LIN {X 0,Y 467.594,Z 130.241,A -85,B 0,C 180,E1 -7494.888,E2 -7494.888} C_VEL
LIN {X 0,Y 467.619,Z 130.232,A -85,B 0,C 180,E1 -7497.769,E2 -7497.769} C_VEL
LIN {X 0,Y 467.567,Z 130.241,A -85,B 0,C 180,E1 -7501.045,E2 -7501.045} C_VEL
LIN {X 0,Y 467.576,Z 130.242,A -85,B 0,C 180,E1 -7504.24,E2 -7504.24} C_VEL
LIN {X 0,Y 467.547,Z 130.241,A -85,B 0,C 180,E1 -7507.186,E2 -7507.186} C_VEL
LIN {X 0,Y 467.573,Z 130.245,A -85,B 0,C 180,E1 -7510.265,E2 -7510.265} C_VEL
LIN {X 0,Y 467.585,Z 130.24,A -85,B 0,C 180,E1 -7512.567,E2 -7512.567} C_VEL
LIN {X 0,Y 467.569,Z 130.238,A -85,B 0,C 180,E1 -7515.053,E2 -7515.053} C_VEL
LIN {X 0,Y 467.587,Z 130.236,A -85,B 0,C 180,E1 -7517.44,E2 -7517.44} C_VEL
LIN {X 0,Y 467.581,Z 130.237,A -85,B 0,C 180,E1 -7520.855,E2 -7520.855} C_VEL
LIN {X 0,Y 467.56,Z 130.244,A -85,B 0,C 180,E1 -7524.26,E2 -7524.26} C_VEL
LIN {X 0,Y 467.58,Z 130.238,A -85,B 0,C 180,E1 -7527.321,E2 -7527.321} C_VEL
LIN {X 0,Y 467.569,Z 130.238,A -85,B 0,C 180,E1 -7530.667,E2 -7530.667} C_VEL
LIN {X 0,Y 467.611,Z 130.234,A -85,B 0,C 180,E1 -7533.2,E2 -7533.2} C_VEL
LIN {X 0,Y 467.588,Z 130.236,A -85,B 0,C 180,E1 -7536.469,E2 -7536.469} C_VEL
LIN {X 0,Y 467.621,Z 130.237,A -85,B 0,C 180,E1 -7539.777,E2 -7539.777} C_VEL
LIN {X 0,Y 467.607,Z 130.233,A -85,B 0,C 180,E1 -7542.507,E2 -7542.507} C_VEL
LIN {X 0,Y 467.608,Z 130.238,A -85,B 0,C 180,E1 -7545.197,E2 -7545.197} C_VEL
LIN {X 0,Y 467.654,Z 130.23,A -85,B 0,C 180,E1 -7547.855,E2 -7547.855} C_VEL
LIN {X 0,Y 467.68,Z 130.232,A -85,B 0,C 180,E1 -7551.357,E2 -7551.357} C_VEL
LIN {X 0,Y 467.744,Z 130.217,A -85,B 0,C 180,E1 -7553.963,E2 -7553.963} C_VEL
LIN {X 0,Y 467.858,Z 130.207,A -85,B 0,C 180,E1 -7557.417,E2 -7557.417} C_VEL
LIN {X 0,Y 467.881,Z 130.199,A -85,B 0,C 180,E1 -7560,E2 -7560} C_VEL
LIN {X 0,Y 467.858,Z 130.204,A -85,B 0,C 180,E1 -7562.583,E2 -7562.583} C_VEL
LIN {X 0,Y 467.734,Z 130.218,A -85,B 0,C 180,E1 -7566.038,E2 -7566.038} C_VEL
LIN {X 0,Y 467.68,Z 130.229,A -85,B 0,C 180,E1 -7568.643,E2 -7568.643} C_VEL
LIN {X 0,Y 467.655,Z 130.228,A -85,B 0,C 180,E1 -7572.146,E2 -7572.146} C_VEL
LIN {X 0,Y 467.638,Z 130.229,A -85,B 0,C 180,E1 -7575.695,E2 -7575.695} C_VEL
LIN {X 0,Y 467.617,Z 130.238,A -85,B 0,C 180,E1 -7578.765,E2 -7578.765} C_VEL
LIN {X 0,Y 467.579,Z 130.238,A -85,B 0,C 180,E1 -7581.268,E2 -7581.268} C_VEL
LIN {X 0,Y 467.571,Z 130.239,A -85,B 0,C 180,E1 -7583.944,E2 -7583.944} C_VEL
LIN {X 0,Y 467.616,Z 130.236,A -85,B 0,C 180,E1 -7586.801,E2 -7586.801} C_VEL
LIN {X 0,Y 467.553,Z 130.241,A -85,B 0,C 180,E1 -7589.738,E2 -7589.738} C_VEL
LIN {X 0,Y 467.583,Z 130.239,A -85,B 0,C 180,E1 -7592.759,E2 -7592.759} C_VEL
LIN {X 0,Y 467.553,Z 130.244,A -85,B 0,C 180,E1 -7595.89,E2 -7595.89} C_VEL
LIN {X 0,Y 467.6,Z 130.234,A -85,B 0,C 180,E1 -7599.143,E2 -7599.143} C_VEL
LIN {X 0,Y 467.587,Z 130.238,A -85,B 0,C 180,E1 -7602.567,E2 -7602.567} C_VEL
LIN {X 0,Y 467.571,Z 130.238,A -85,B 0,C 180,E1 -7605.053,E2 -7605.053} C_VEL
LIN {X 0,Y 467.59,Z 130.238,A -85,B 0,C 180,E1 -7607.44,E2 -7607.44} C_VEL
LIN {X 0,Y 467.601,Z 130.234,A -85,B 0,C 180,E1 -7610.857,E2 -7610.857} C_VEL
LIN {X 0,Y 467.561,Z 130.241,A -85,B 0,C 180,E1 -7614.261,E2 -7614.261} C_VEL
LIN {X 0,Y 467.583,Z 130.24,A -85,B 0,C 180,E1 -7617.321,E2 -7617.321} C_VEL
LIN {X 0,Y 467.572,Z 130.242,A -85,B 0,C 180,E1 -7620.668,E2 -7620.668} C_VEL
LIN {X 0,Y 467.701,Z 130.331,A -85,B 0,C 180,E1 -7623.093,E2 -7623.093} C_VEL
LIN {X 0,Y 470,Z 142.281,A -85,B 0,C 180,E1 -7625.248,E2 -7625.248} C_VEL
LIN {X 0,Y 469.567,Z 154.773,A -85,B 0,C 180,E1 -7627.332,E2 -7627.332} C_VEL
LIN {X 0,Y 468.805,Z 175.972,A -85,B 0,C 180,E1 -7630.814,E2 -7630.814} C_VEL
LIN {X 0,Y 468.241,Z 189.54,A -85,B 0,C 180,E1 -7633.002,E2 -7633.002} C_VEL
LIN {X 0,Y 471.063,Z 210.719,A -85,B 0,C 180,E1 -7633.441,E2 -7633.441} C_VEL
LIN {X 0,Y 470.388,Z 298.839,A -85,B 0,C 180,E1 -7634.843,E2 -7634.843} C_VEL
LIN {X 0,Y 469.978,Z 311.849,A -85,B 0,C 180,E1 -7635.218,E2 -7635.218} C_VEL
LIN {X 0,Y 469.486,Z 324.472,A -85,B 0,C 180,E1 -7635.755,E2 -7635.755} C_VEL
LIN {X 0,Y 469.009,Z 336.521,A -85,B 0,C 180,E1 -7636.459,E2 -7636.459} C_VEL
LIN {X 0,Y 468.479,Z 348.326,A -85,B 0,C 180,E1 -7637.35,E2 -7637.35} C_VEL
LIN {X 0,Y 468.04,Z 358.45,A -85,B 0,C 180,E1 -7638.304,E2 -7638.304} C_VEL
LIN {X 0,Y 467.56,Z 367.788,A -85,B 0,C 180,E1 -7639.389,E2 -7639.389} C_VEL
LIN {X 0,Y 467.188,Z 376.856,A -85,B 0,C 180,E1 -7640.694,E2 -7640.694} C_VEL
LIN {X 0,Y 466.977,Z 384.164,A -85,B 0,C 180,E1 -7641.998,E2 -7641.998} C_VEL
LIN {X 0,Y 466.827,Z 389.097,A -85,B 0,C 180,E1 -7643.083,E2 -7643.083} C_VEL
LIN {X 0,Y 466.746,Z 393.889,A -85,B 0,C 180,E1 -7644.383,E2 -7644.383} C_VEL
LIN {X 0,Y 466.659,Z 397.547,A -85,B 0,C 180,E1 -7645.681,E2 -7645.681} C_VEL
LIN {X 0,Y 466.747,Z 399.441,A -85,B 0,C 180,E1 -7646.547,E2 -7646.547} C_VEL
LIN {X 0,Y 466.711,Z 400.855,A -85,B 0,C 180,E1 -7647.411,E2 -7647.411} C_VEL
LIN {X 0,Y 466.696,Z 401.858,A -85,B 0,C 180,E1 -7648.274,E2 -7648.274} C_VEL
LIN {X 0,Y 466.621,Z 402.678,A -85,B 0,C 180,E1 -7650,E2 -7650} C_VEL
LIN {X 0,Y 466.634,Z 402.453,A -85,B 0,C 180,E1 -7650.863,E2 -7650.863} C_VEL
LIN {X 0,Y 466.696,Z 401.831,A -85,B 0,C 180,E1 -7651.726,E2 -7651.726} C_VEL
LIN {X 0,Y 466.711,Z 400.812,A -85,B 0,C 180,E1 -7652.589,E2 -7652.589} C_VEL
LIN {X 0,Y 466.748,Z 399.388,A -85,B 0,C 180,E1 -7653.453,E2 -7653.453} C_VEL
LIN {X 0,Y 466.689,Z 396.392,A -85,B 0,C 180,E1 -7654.751,E2 -7654.751} C_VEL
LIN {X 0,Y 466.713,Z 392.348,A -85,B 0,C 180,E1 -7656.051,E2 -7656.051} C_VEL
LIN {X 0,Y 466.904,Z 386.14,A -85,B 0,C 180,E1 -7657.568,E2 -7657.568} C_VEL
LIN {X 0,Y 467.077,Z 379.359,A -85,B 0,C 180,E1 -7658.872,E2 -7658.872} C_VEL
LIN {X 0,Y 467.396,Z 370.96,A -85,B 0,C 180,E1 -7660.176,E2 -7660.176} C_VEL
LIN {X 0,Y 467.834,Z 362.352,A -85,B 0,C 180,E1 -7661.262,E2 -7661.262} C_VEL
LIN {X 0,Y 468.252,Z 352.515,A -85,B 0,C 180,E1 -7662.277,E2 -7662.277} C_VEL
LIN {X 0,Y 468.773,Z 341.227,A -85,B 0,C 180,E1 -7663.216,E2 -7663.216} C_VEL
LIN {X 0,Y 469.307,Z 329.707,A -85,B 0,C 180,E1 -7663.974,E2 -7663.974} C_VEL
LIN {X 0,Y 469.764,Z 317.81,A -85,B 0,C 180,E1 -7664.568,E2 -7664.568} C_VEL
LIN {X 0,Y 470.275,Z 304.132,A -85,B 0,C 180,E1 -7665.05,E2 -7665.05} C_VEL
LIN {X 0,Y 470.563,Z 290.188,A -85,B 0,C 180,E1 -7665.345,E2 -7665.345} C_VEL
LIN {X 0,Y 471.015,Z 208.612,A -85,B 0,C 180,E1 -7666.634,E2 -7666.634} C_VEL
LIN {X 0,Y 468.224,Z 188.606,A -85,B 0,C 180,E1 -7667.064,E2 -7667.064} C_VEL
LIN {X 0,Y 468.823,Z 169.364,A -85,B 0,C 180,E1 -7670.169,E2 -7670.169} C_VEL
LIN {X 0,Y 469.527,Z 152.566,A -85,B 0,C 180,E1 -7672.903,E2 -7672.903} C_VEL
LIN {X 0,Y 469.89,Z 142.442,A -85,B 0,C 180,E1 -7674.575,E2 -7674.575} C_VEL
LIN {X 0,Y 468.192,Z 132.826,A -85,B 0,C 180,E1 -7676.283,E2 -7676.283} C_VEL
LIN {X 0,Y 467.673,Z 130.234,A -85,B 0,C 180,E1 -7676.797,E2 -7676.797} C_VEL
LIN {X 0,Y 467.556,Z 130.246,A -85,B 0,C 180,E1 -7679.738,E2 -7679.738} C_VEL
LIN {X 0,Y 467.584,Z 130.242,A -85,B 0,C 180,E1 -7682.758,E2 -7682.758} C_VEL
LIN {X 0,Y 467.554,Z 130.246,A -85,B 0,C 180,E1 -7685.889,E2 -7685.889} C_VEL
LIN {X 0,Y 467.601,Z 130.238,A -85,B 0,C 180,E1 -7689.143,E2 -7689.143} C_VEL
LIN {X 0,Y 467.587,Z 130.241,A -85,B 0,C 180,E1 -7692.567,E2 -7692.567} C_VEL
LIN {X 0,Y 467.57,Z 130.241,A -85,B 0,C 180,E1 -7695.053,E2 -7695.053} C_VEL
LIN {X 0,Y 467.589,Z 130.24,A -85,B 0,C 180,E1 -7697.44,E2 -7697.44} C_VEL
LIN {X 0,Y 467.599,Z 130.234,A -85,B 0,C 180,E1 -7700.857,E2 -7700.857} C_VEL
LIN {X 0,Y 467.559,Z 130.243,A -85,B 0,C 180,E1 -7704.261,E2 -7704.261} C_VEL
LIN {X 0,Y 467.581,Z 130.238,A -85,B 0,C 180,E1 -7707.321,E2 -7707.321} C_VEL
LIN {X 0,Y 467.568,Z 130.236,A -85,B 0,C 180,E1 -7710.667,E2 -7710.667} C_VEL
LIN {X 0,Y 467.612,Z 130.235,A -85,B 0,C 180,E1 -7713.199,E2 -7713.199} C_VEL
LIN {X 0,Y 467.589,Z 130.234,A -85,B 0,C 180,E1 -7716.468,E2 -7716.468} C_VEL
LIN {X 0,Y 467.622,Z 130.234,A -85,B 0,C 180,E1 -7719.777,E2 -7719.777} C_VEL
LIN {X 0,Y 467.607,Z 130.233,A -85,B 0,C 180,E1 -7722.506,E2 -7722.506} C_VEL
LIN {X 0,Y 467.608,Z 130.235,A -85,B 0,C 180,E1 -7725.196,E2 -7725.196} C_VEL
LIN {X 0,Y 467.654,Z 130.228,A -85,B 0,C 180,E1 -7727.854,E2 -7727.854} C_VEL
LIN {X 0,Y 467.68,Z 130.229,A -85,B 0,C 180,E1 -7731.357,E2 -7731.357} C_VEL
LIN {X 0,Y 467.744,Z 130.218,A -85,B 0,C 180,E1 -7733.962,E2 -7733.962} C_VEL
LIN {X 0,Y 467.858,Z 130.207,A -85,B 0,C 180,E1 -7737.417,E2 -7737.417} C_VEL
LIN {X 0,Y 467.881,Z 130.198,A -85,B 0,C 180,E1 -7740,E2 -7740} C_VEL
LIN {X 0,Y 467.858,Z 130.206,A -85,B 0,C 180,E1 -7742.583,E2 -7742.583} C_VEL
LIN {X 0,Y 467.733,Z 130.217,A -85,B 0,C 180,E1 -7746.037,E2 -7746.037} C_VEL
LIN {X 0,Y 467.679,Z 130.231,A -85,B 0,C 180,E1 -7748.643,E2 -7748.643} C_VEL
LIN {X 0,Y 467.654,Z 130.229,A -85,B 0,C 180,E1 -7752.145,E2 -7752.145} C_VEL
LIN {X 0,Y 467.637,Z 130.231,A -85,B 0,C 180,E1 -7755.695,E2 -7755.695} C_VEL
LIN {X 0,Y 467.615,Z 130.24,A -85,B 0,C 180,E1 -7758.765,E2 -7758.765} C_VEL
LIN {X 0,Y 467.578,Z 130.239,A -85,B 0,C 180,E1 -7761.268,E2 -7761.268} C_VEL
LIN {X 0,Y 467.569,Z 130.244,A -85,B 0,C 180,E1 -7763.943,E2 -7763.943} C_VEL
LIN {X 0,Y 467.614,Z 130.24,A -85,B 0,C 180,E1 -7766.8,E2 -7766.8} C_VEL
LIN {X 0,Y 467.552,Z 130.244,A -85,B 0,C 180,E1 -7769.738,E2 -7769.738} C_VEL
LIN {X 0,Y 467.582,Z 130.244,A -85,B 0,C 180,E1 -7772.758,E2 -7772.758} C_VEL
LIN {X 0,Y 467.651,Z 130.325,A -85,B 0,C 180,E1 -7773.589,E2 -7773.589} C_VEL
LIN {X 0,Y 468.729,Z 136.861,A -85,B 0,C 180,E1 -7774.995,E2 -7774.995} C_VEL
LIN {X 0,Y 468.69,Z 141.798,A -85,B 0,C 180,E1 -7776.011,E2 -7776.011} C_VEL
LIN {X 0,Y 471.496,Z 154.916,A -85,B 0,C 180,E1 -7776.345,E2 -7776.345} C_VEL
LIN {X 0,Y 470.667,Z 248.936,A -85,B 0,C 180,E1 -7777.851,E2 -7777.851} C_VEL
LIN {X 0,Y 470.374,Z 262.577,A -85,B 0,C 180,E1 -7778.252,E2 -7778.252} C_VEL
LIN {X 0,Y 470.103,Z 274.187,A -85,B 0,C 180,E1 -7778.757,E2 -7778.757} C_VEL
LIN {X 0,Y 469.739,Z 285.551,A -85,B 0,C 180,E1 -7779.414,E2 -7779.414} C_VEL
LIN {X 0,Y 469.285,Z 296.959,A -85,B 0,C 180,E1 -7780.267,E2 -7780.267} C_VEL
LIN {X 0,Y 468.755,Z 307.729,A -85,B 0,C 180,E1 -7781.276,E2 -7781.276} C_VEL
LIN {X 0,Y 468.315,Z 316.44,A -85,B 0,C 180,E1 -7782.282,E2 -7782.282} C_VEL
LIN {X 0,Y 467.855,Z 325.055,A -85,B 0,C 180,E1 -7783.503,E2 -7783.503} C_VEL
LIN {X 0,Y 467.497,Z 332.108,A -85,B 0,C 180,E1 -7784.737,E2 -7784.737} C_VEL
LIN {X 0,Y 467.196,Z 338.877,A -85,B 0,C 180,E1 -7786.225,E2 -7786.225} C_VEL
LIN {X 0,Y 467.002,Z 343.41,A -85,B 0,C 180,E1 -7787.511,E2 -7787.511} C_VEL
LIN {X 0,Y 466.836,Z 346.943,A -85,B 0,C 180,E1 -7788.827,E2 -7788.827} C_VEL
LIN {X 0,Y 466.724,Z 349.492,A -85,B 0,C 180,E1 -7790.171,E2 -7790.171} C_VEL
LIN {X 0,Y 466.622,Z 351.29,A -85,B 0,C 180,E1 -7791.919,E2 -7791.919} C_VEL
LIN {X 0,Y 466.617,Z 351.63,A -85,B 0,C 180,E1 -7792.964,E2 -7792.964} C_VEL
LIN {X 0,Y 466.608,Z 351.1,A -85,B 0,C 180,E1 -7794.424,E2 -7794.424} C_VEL
LIN {X 0,Y 466.69,Z 349.689,A -85,B 0,C 180,E1 -7795.672,E2 -7795.672} C_VEL
LIN {X 0,Y 466.103,Z 348.636,A -85,B 0,C 180,E1 -7796.383,E2 -7796.383} C_VEL
LIN {X 0,Y 463.361,Z 346.465,A -85,B 0,C 180,E1 -7797.529,E2 -7797.529} C_VEL
LIN {X 0,Y 461.039,Z 344.188,A -85,B 0,C 180,E1 -7798.432,E2 -7798.432} C_VEL
LIN {X 0,Y 460.075,Z 342.059,A -85,B 0,C 180,E1 -7799.112,E2 -7799.112} C_VEL
LIN {X 0,Y 460.016,Z 341.258,A -85,B 0,C 180,E1 -7799.338,E2 -7799.338} C_VEL
LIN {X 0,Y 460.283,Z 335.541,A -85,B 0,C 180,E1 -7800.751,E2 -7800.751} C_VEL
LIN {X 0,Y 460.683,Z 327.924,A -85,B 0,C 180,E1 -7802.23,E2 -7802.23} C_VEL
LIN {X 0,Y 461.124,Z 319.458,A -85,B 0,C 180,E1 -7803.526,E2 -7803.526} C_VEL
LIN {X 0,Y 461.649,Z 309.352,A -85,B 0,C 180,E1 -7804.77,E2 -7804.77} C_VEL
LIN {X 0,Y 462.112,Z 299.402,A -85,B 0,C 180,E1 -7805.756,E2 -7805.756} C_VEL
LIN {X 0,Y 462.609,Z 288.553,A -85,B 0,C 180,E1 -7806.616,E2 -7806.616} C_VEL
LIN {X 0,Y 463.013,Z 276.885,A -85,B 0,C 180,E1 -7807.346,E2 -7807.346} C_VEL
LIN {X 0,Y 463.364,Z 265.358,A -85,B 0,C 180,E1 -7807.894,E2 -7807.894} C_VEL
LIN {X 0,Y 463.657,Z 252.665,A -85,B 0,C 180,E1 -7808.317,E2 -7808.317} C_VEL
LIN {X 0,Y 463.828,Z 237.232,A -85,B 0,C 180,E1 -7808.617,E2 -7808.617} C_VEL
LIN {X 0,Y 464.471,Z 155.674,A -85,B 0,C 180,E1 -7809.919,E2 -7809.919} C_VEL
LIN {X 0,Y 461.531,Z 141.472,A -85,B 0,C 180,E1 -7810.279,E2 -7810.279} C_VEL
LIN {X 0,Y 461.356,Z 135.46,A -85,B 0,C 180,E1 -7811.573,E2 -7811.573} C_VEL
LIN {X 0,Y 460.578,Z 131.114,A -85,B 0,C 180,E1 -7812.575,E2 -7812.575} C_VEL
LIN {X 0,Y 460.565,Z 131.114,A -85,B 0,C 180,E1 -7814.965,E2 -7814.965} C_VEL
LIN {X 0,Y 460.61,Z 131.105,A -85,B 0,C 180,E1 -7818.559,E2 -7818.559} C_VEL
LIN {X 0,Y 460.695,Z 131.096,A -85,B 0,C 180,E1 -7822.109,E2 -7822.109} C_VEL
LIN {X 0,Y 460.695,Z 131.095,A -85,B 0,C 180,E1 -7824.748,E2 -7824.748} C_VEL
LIN {X 0,Y 460.799,Z 131.089,A -85,B 0,C 180,E1 -7827.378,E2 -7827.378} C_VEL
LIN {X 0,Y 460.853,Z 131.076,A -85,B 0,C 180,E1 -7830,E2 -7830} C_VEL
LIN {X 0,Y 460.8,Z 131.082,A -85,B 0,C 180,E1 -7832.623,E2 -7832.623} C_VEL
LIN {X 0,Y 460.688,Z 131.095,A -85,B 0,C 180,E1 -7836.13,E2 -7836.13} C_VEL
LIN {X 0,Y 460.619,Z 131.107,A -85,B 0,C 180,E1 -7838.776,E2 -7838.776} C_VEL
LIN {X 0,Y 460.614,Z 131.106,A -85,B 0,C 180,E1 -7842.445,E2 -7842.445} C_VEL
LIN {X 0,Y 460.6,Z 131.106,A -85,B 0,C 180,E1 -7845.997,E2 -7845.997} C_VEL
LIN {X 0,Y 460.568,Z 131.111,A -85,B 0,C 180,E1 -7849.615,E2 -7849.615} C_VEL
LIN {X 0,Y 460.51,Z 131.121,A -85,B 0,C 180,E1 -7852.429,E2 -7852.429} C_VEL
LIN {X 0,Y 460.557,Z 131.112,A -85,B 0,C 180,E1 -7855.799,E2 -7855.799} C_VEL
LIN {X 0,Y 460.552,Z 131.115,A -85,B 0,C 180,E1 -7858.233,E2 -7858.233} C_VEL
LIN {X 0,Y 460.519,Z 131.117,A -85,B 0,C 180,E1 -7861.283,E2 -7861.283} C_VEL
LIN {X 0,Y 460.522,Z 131.124,A -85,B 0,C 180,E1 -7864.504,E2 -7864.504} C_VEL
LIN {X 0,Y 460.5,Z 131.119,A -85,B 0,C 180,E1 -7867.623,E2 -7867.623} C_VEL
LIN {X 0,Y 460.537,Z 131.121,A -85,B 0,C 180,E1 -7870.269,E2 -7870.269} C_VEL
LIN {X 0,Y 460.498,Z 131.119,A -85,B 0,C 180,E1 -7873.375,E2 -7873.375} C_VEL
LIN {X 0,Y 460.498,Z 131.122,A -85,B 0,C 180,E1 -7876.625,E2 -7876.625} C_VEL
LIN {X 0,Y 460.54,Z 131.117,A -85,B 0,C 180,E1 -7879.731,E2 -7879.731} C_VEL
LIN {X 0,Y 460.525,Z 131.118,A -85,B 0,C 180,E1 -7882.519,E2 -7882.519} C_VEL
LIN {X 0,Y 460.546,Z 131.117,A -85,B 0,C 180,E1 -7885.624,E2 -7885.624} C_VEL
LIN {X 0,Y 460.535,Z 131.114,A -85,B 0,C 180,E1 -7888.745,E2 -7888.745} C_VEL
LIN {X 0,Y 460.579,Z 131.111,A -85,B 0,C 180,E1 -7892.254,E2 -7892.254} C_VEL
LIN {X 0,Y 460.537,Z 131.114,A -85,B 0,C 180,E1 -7894.704,E2 -7894.704} C_VEL
LIN {X 0,Y 460.508,Z 131.124,A -85,B 0,C 180,E1 -7897.571,E2 -7897.571} C_VEL
LIN {X 0,Y 460.567,Z 131.111,A -85,B 0,C 180,E1 -7900.385,E2 -7900.385} C_VEL
LIN {X 0,Y 460.563,Z 131.114,A -85,B 0,C 180,E1 -7903.146,E2 -7903.146} C_VEL
LIN {X 0,Y 460.556,Z 131.115,A -85,B 0,C 180,E1 -7905.868,E2 -7905.868} C_VEL
LIN {X 0,Y 460.61,Z 131.105,A -85,B 0,C 180,E1 -7908.559,E2 -7908.559} C_VEL
LIN {X 0,Y 460.694,Z 131.095,A -85,B 0,C 180,E1 -7912.109,E2 -7912.109} C_VEL
LIN {X 0,Y 460.697,Z 131.096,A -85,B 0,C 180,E1 -7914.749,E2 -7914.749} C_VEL
LIN {X 0,Y 460.823,Z 131.084,A -85,B 0,C 180,E1 -7917.378,E2 -7917.378} C_VEL
LIN {X 0,Y 460.852,Z 131.075,A -85,B 0,C 180,E1 -7920,E2 -7920} C_VEL
LIN {X 0,Y 460.823,Z 131.081,A -85,B 0,C 180,E1 -7922.623,E2 -7922.623} C_VEL
LIN {X 0,Y 460.7,Z 131.094,A -85,B 0,C 180,E1 -7926.13,E2 -7926.13} C_VEL
LIN {X 0,Y 460.627,Z 131.109,A -85,B 0,C 180,E1 -7928.776,E2 -7928.776} C_VEL
LIN {X 0,Y 460.612,Z 131.108,A -85,B 0,C 180,E1 -7932.445,E2 -7932.445} C_VEL
LIN {X 0,Y 460.599,Z 131.107,A -85,B 0,C 180,E1 -7935.998,E2 -7935.998} C_VEL
LIN {X 0,Y 460.57,Z 131.114,A -85,B 0,C 180,E1 -7938.902,E2 -7938.902} C_VEL
LIN {X 0,Y 460.515,Z 131.117,A -85,B 0,C 180,E1 -7941.486,E2 -7941.486} C_VEL
LIN {X 0,Y 460.541,Z 131.119,A -85,B 0,C 180,E1 -7944.333,E2 -7944.333} C_VEL
LIN {X 0,Y 460.572,Z 131.11,A -85,B 0,C 180,E1 -7947.244,E2 -7947.244} C_VEL
LIN {X 0,Y 460.51,Z 131.124,A -85,B 0,C 180,E1 -7950.24,E2 -7950.24} C_VEL
LIN {X 0,Y 460.529,Z 131.115,A -85,B 0,C 180,E1 -7953.325,E2 -7953.325} C_VEL
LIN {X 0,Y 460.476,Z 131.125,A -85,B 0,C 180,E1 -7956.53,E2 -7956.53} C_VEL
LIN {X 0,Y 460.575,Z 131.114,A -85,B 0,C 180,E1 -7959.858,E2 -7959.858} C_VEL
LIN {X 0,Y 460.513,Z 131.117,A -85,B 0,C 180,E1 -7962.901,E2 -7962.901} C_VEL
LIN {X 0,Y 460.512,Z 131.123,A -85,B 0,C 180,E1 -7965.831,E2 -7965.831} C_VEL
LIN {X 0,Y 460.54,Z 131.114,A -85,B 0,C 180,E1 -7968.99,E2 -7968.99} C_VEL
LIN {X 0,Y 460.541,Z 131.115,A -85,B 0,C 180,E1 -7971.269,E2 -7971.269} C_VEL
LIN {X 0,Y 460.511,Z 131.117,A -85,B 0,C 180,E1 -7974.555,E2 -7974.555} C_VEL
LIN {X 0,Y 460.533,Z 131.122,A -85,B 0,C 180,E1 -7977.716,E2 -7977.716} C_VEL
LIN {X 0,Y 460.542,Z 131.118,A -85,B 0,C 180,E1 -7980.769,E2 -7980.769} C_VEL
LIN {X 0,Y 460.66,Z 131.23,A -85,B 0,C 180,E1 -7982.885,E2 -7982.885} C_VEL
LIN {X 0,Y 463.022,Z 143.219,A -85,B 0,C 180,E1 -7985.086,E2 -7985.086} C_VEL
LIN {X 0,Y 462.816,Z 151.577,A -85,B 0,C 180,E1 -7986.509,E2 -7986.509} C_VEL
LIN {X 0,Y 462.035,Z 168.201,A -85,B 0,C 180,E1 -7989.289,E2 -7989.289} C_VEL
LIN {X 0,Y 461.526,Z 182.026,A -85,B 0,C 180,E1 -7991.58,E2 -7991.58} C_VEL
LIN {X 0,Y 461.248,Z 189.092,A -85,B 0,C 180,E1 -7992.743,E2 -7992.743} C_VEL
LIN {X 0,Y 464.245,Z 211.74,A -85,B 0,C 180,E1 -7993.221,E2 -7993.221} C_VEL
LIN {X 0,Y 463.532,Z 297.985,A -85,B 0,C 180,E1 -7994.613,E2 -7994.613} C_VEL
LIN {X 0,Y 463.111,Z 311.151,A -85,B 0,C 180,E1 -7994.993,E2 -7994.993} C_VEL
LIN {X 0,Y 462.596,Z 323.858,A -85,B 0,C 180,E1 -7995.539,E2 -7995.539} C_VEL
LIN {X 0,Y 462.055,Z 335.978,A -85,B 0,C 180,E1 -7996.252,E2 -7996.252} C_VEL
LIN {X 0,Y 461.486,Z 347.816,A -85,B 0,C 180,E1 -7997.155,E2 -7997.155} C_VEL
LIN {X 0,Y 461.023,Z 357.967,A -85,B 0,C 180,E1 -7998.124,E2 -7998.124} C_VEL
LIN {X 0,Y 460.557,Z 367.336,A -85,B 0,C 180,E1 -7999.226,E2 -7999.226} C_VEL
LIN {X 0,Y 460.142,Z 376.418,A -85,B 0,C 180,E1 -8000.55,E2 -8000.55} C_VEL
LIN {X 0,Y 459.903,Z 383.737,A -85,B 0,C 180,E1 -8001.874,E2 -8001.874} C_VEL
LIN {X 0,Y 459.74,Z 388.679,A -85,B 0,C 180,E1 -8002.975,E2 -8002.975} C_VEL
LIN {X 0,Y 459.642,Z 393.478,A -85,B 0,C 180,E1 -8004.296,E2 -8004.296} C_VEL
LIN {X 0,Y 459.575,Z 397.145,A -85,B 0,C 180,E1 -8005.615,E2 -8005.615} C_VEL
LIN {X 0,Y 459.642,Z 399.041,A -85,B 0,C 180,E1 -8006.494,E2 -8006.494} C_VEL
LIN {X 0,Y 459.631,Z 400.461,A -85,B 0,C 180,E1 -8007.371,E2 -8007.371} C_VEL
LIN {X 0,Y 459.617,Z 401.467,A -85,B 0,C 180,E1 -8008.247,E2 -8008.247} C_VEL
LIN {X 0,Y 459.551,Z 402.29,A -85,B 0,C 180,E1 -8010,E2 -8010} C_VEL
LIN {X 0,Y 459.566,Z 402.068,A -85,B 0,C 180,E1 -8010.876,E2 -8010.876} C_VEL
LIN {X 0,Y 459.604,Z 401.444,A -85,B 0,C 180,E1 -8011.752,E2 -8011.752} C_VEL
LIN {X 0,Y 459.631,Z 400.426,A -85,B 0,C 180,E1 -8012.629,E2 -8012.629} C_VEL
LIN {X 0,Y 459.642,Z 399.001,A -85,B 0,C 180,E1 -8013.506,E2 -8013.506} C_VEL
LIN {X 0,Y 459.619,Z 396.006,A -85,B 0,C 180,E1 -8014.824,E2 -8014.824} C_VEL
LIN {X 0,Y 459.635,Z 391.248,A -85,B 0,C 180,E1 -8016.342,E2 -8016.342} C_VEL
LIN {X 0,Y 459.865,Z 384.729,A -85,B 0,C 180,E1 -8017.906,E2 -8017.906} C_VEL
LIN {X 0,Y 460.086,Z 377.725,A -85,B 0,C 180,E1 -8019.23,E2 -8019.23} C_VEL
LIN {X 0,Y 460.442,Z 368.969,A -85,B 0,C 180,E1 -8020.554,E2 -8020.554} C_VEL
LIN {X 0,Y 460.95,Z 360.009,A -85,B 0,C 180,E1 -8021.655,E2 -8021.655} C_VEL
LIN {X 0,Y 461.436,Z 349.203,A -85,B 0,C 180,E1 -8022.738,E2 -8022.738} C_VEL
LIN {X 0,Y 461.969,Z 337.843,A -85,B 0,C 180,E1 -8023.639,E2 -8023.639} C_VEL
LIN {X 0,Y 462.586,Z 325.398,A -85,B 0,C 180,E1 -8024.405,E2 -8024.405} C_VEL
LIN {X 0,Y 463.06,Z 313.6,A -85,B 0,C 180,E1 -8024.952,E2 -8024.952} C_VEL
LIN {X 0,Y 463.512,Z 300.871,A -85,B 0,C 180,E1 -8025.359,E2 -8025.359} C_VEL
LIN {X 0,Y 463.773,Z 283.141,A -85,B 0,C 180,E1 -8025.688,E2 -8025.688} C_VEL
LIN {X 0,Y 464.2,Z 209.161,A -85,B 0,C 180,E1 -8026.879,E2 -8026.879} C_VEL
LIN {X 0,Y 461.246,Z 188.093,A -85,B 0,C 180,E1 -8027.356,E2 -8027.356} C_VEL
LIN {X 0,Y 461.892,Z 169.002,A -85,B 0,C 180,E1 -8030.485,E2 -8030.485} C_VEL
LIN {X 0,Y 462.645,Z 152.228,A -85,B 0,C 180,E1 -8033.263,E2 -8033.263} C_VEL
LIN {X 0,Y 462.968,Z 143.686,A -85,B 0,C 180,E1 -8034.698,E2 -8034.698} C_VEL
LIN {X 0,Y 461.199,Z 133.885,A -85,B 0,C 180,E1 -8036.47,E2 -8036.47} C_VEL
LIN {X 0,Y 460.638,Z 131.109,A -85,B 0,C 180,E1 -8036.994,E2 -8036.994} C_VEL
LIN {X 0,Y 460.512,Z 131.125,A -85,B 0,C 180,E1 -8040.24,E2 -8040.24} C_VEL
LIN {X 0,Y 460.53,Z 131.118,A -85,B 0,C 180,E1 -8043.324,E2 -8043.324} C_VEL
LIN {X 0,Y 460.477,Z 131.129,A -85,B 0,C 180,E1 -8046.529,E2 -8046.529} C_VEL
LIN {X 0,Y 460.575,Z 131.117,A -85,B 0,C 180,E1 -8049.857,E2 -8049.857} C_VEL
LIN {X 0,Y 460.513,Z 131.12,A -85,B 0,C 180,E1 -8052.9,E2 -8052.9} C_VEL
LIN {X 0,Y 460.512,Z 131.124,A -85,B 0,C 180,E1 -8055.83,E2 -8055.83} C_VEL
LIN {X 0,Y 460.539,Z 131.115,A -85,B 0,C 180,E1 -8058.989,E2 -8058.989} C_VEL
LIN {X 0,Y 460.539,Z 131.114,A -85,B 0,C 180,E1 -8061.268,E2 -8061.268} C_VEL
LIN {X 0,Y 460.509,Z 131.119,A -85,B 0,C 180,E1 -8064.554,E2 -8064.554} C_VEL
LIN {X 0,Y 460.53,Z 131.119,A -85,B 0,C 180,E1 -8067.715,E2 -8067.715} C_VEL
LIN {X 0,Y 460.538,Z 131.112,A -85,B 0,C 180,E1 -8070.769,E2 -8070.769} C_VEL
LIN {X 0,Y 460.555,Z 131.115,A -85,B 0,C 180,E1 -8073.734,E2 -8073.734} C_VEL
LIN {X 0,Y 460.543,Z 131.112,A -85,B 0,C 180,E1 -8076.624,E2 -8076.624} C_VEL
LIN {X 0,Y 460.551,Z 131.118,A -85,B 0,C 180,E1 -8079.453,E2 -8079.453} C_VEL
LIN {X 0,Y 460.558,Z 131.111,A -85,B 0,C 180,E1 -8082.23,E2 -8082.23} C_VEL
LIN {X 0,Y 460.566,Z 131.111,A -85,B 0,C 180,E1 -8084.965,E2 -8084.965} C_VEL
LIN {X 0,Y 460.61,Z 131.104,A -85,B 0,C 180,E1 -8088.559,E2 -8088.559} C_VEL
LIN {X 0,Y 460.693,Z 131.093,A -85,B 0,C 180,E1 -8092.108,E2 -8092.108} C_VEL
LIN {X 0,Y 460.697,Z 131.098,A -85,B 0,C 180,E1 -8094.748,E2 -8094.748} C_VEL
LIN {X 0,Y 460.823,Z 131.084,A -85,B 0,C 180,E1 -8097.377,E2 -8097.377} C_VEL
LIN {X 0,Y 460.851,Z 131.074,A -85,B 0,C 180,E1 -8100,E2 -8100} C_VEL
LIN {X 0,Y 460.823,Z 131.082,A -85,B 0,C 180,E1 -8102.622,E2 -8102.622} C_VEL
LIN {X 0,Y 460.699,Z 131.093,A -85,B 0,C 180,E1 -8106.13,E2 -8106.13} C_VEL
LIN {X 0,Y 460.626,Z 131.109,A -85,B 0,C 180,E1 -8108.776,E2 -8108.776} C_VEL
LIN {X 0,Y 460.611,Z 131.109,A -85,B 0,C 180,E1 -8112.445,E2 -8112.445} C_VEL
LIN {X 0,Y 460.598,Z 131.109,A -85,B 0,C 180,E1 -8115.997,E2 -8115.997} C_VEL
LIN {X 0,Y 460.569,Z 131.116,A -85,B 0,C 180,E1 -8118.902,E2 -8118.902} C_VEL
LIN {X 0,Y 460.513,Z 131.119,A -85,B 0,C 180,E1 -8121.486,E2 -8121.486} C_VEL
LIN {X 0,Y 460.539,Z 131.124,A -85,B 0,C 180,E1 -8124.332,E2 -8124.332} C_VEL
LIN {X 0,Y 460.577,Z 131.114,A -85,B 0,C 180,E1 -8127.243,E2 -8127.243} C_VEL
LIN {X 0,Y 460.509,Z 131.124,A -85,B 0,C 180,E1 -8130.24,E2 -8130.24} C_VEL
LIN {X 0,Y 460.596,Z 131.23,A -85,B 0,C 180,E1 -8133.385,E2 -8133.385} C_VEL
LIN {X 0,Y 461.813,Z 138.418,A -85,B 0,C 180,E1 -8134.95,E2 -8134.95} C_VEL
LIN {X 0,Y 461.772,Z 142.199,A -85,B 0,C 180,E1 -8135.736,E2 -8135.736} C_VEL
LIN {X 0,Y 464.681,Z 155.463,A -85,B 0,C 180,E1 -8136.085,E2 -8136.085} C_VEL
LIN {X 0,Y 463.859,Z 248.684,A -85,B 0,C 180,E1 -8137.6,E2 -8137.6} C_VEL
LIN {X 0,Y 463.563,Z 262.235,A -85,B 0,C 180,E1 -8137.996,E2 -8137.996} C_VEL
LIN {X 0,Y 463.27,Z 274.432,A -85,B 0,C 180,E1 -8138.529,E2 -8138.529} C_VEL
LIN {X 0,Y 462.836,Z 286.618,A -85,B 0,C 180,E1 -8139.248,E2 -8139.248} C_VEL
LIN {X 0,Y 462.386,Z 297.683,A -85,B 0,C 180,E1 -8140.096,E2 -8140.096} C_VEL
LIN {X 0,Y 461.803,Z 308.805,A -85,B 0,C 180,E1 -8141.163,E2 -8141.163} C_VEL
LIN {X 0,Y 461.236,Z 318.639,A -85,B 0,C 180,E1 -8142.353,E2 -8142.353} C_VEL
LIN {X 0,Y 460.795,Z 326.815,A -85,B 0,C 180,E1 -8143.576,E2 -8143.576} C_VEL
LIN {X 0,Y 460.389,Z 334.419,A -85,B 0,C 180,E1 -8144.989,E2 -8144.989} C_VEL
LIN {X 0,Y 460.146,Z 339.707,A -85,B 0,C 180,E1 -8146.224,E2 -8146.224} C_VEL
LIN {X 0,Y 459.9,Z 344.757,A -85,B 0,C 180,E1 -8147.749,E2 -8147.749} C_VEL
LIN {X 0,Y 459.743,Z 347.669,A -85,B 0,C 180,E1 -8148.904,E2 -8148.904} C_VEL
LIN {X 0,Y 459.648,Z 349.763,A -85,B 0,C 180,E1 -8150.046,E2 -8150.046} C_VEL
LIN {X 0,Y 459.566,Z 351.222,A -85,B 0,C 180,E1 -8151.254,E2 -8151.254} C_VEL
LIN {X 0,Y 459.518,Z 351.975,A -85,B 0,C 180,E1 -8152.684,E2 -8152.684} C_VEL
LIN {X 0,Y 459.52,Z 351.464,A -85,B 0,C 180,E1 -8154.467,E2 -8154.467} C_VEL
LIN {X 0,Y 459.615,Z 350.126,A -85,B 0,C 180,E1 -8155.685,E2 -8155.685} C_VEL
LIN {X 0,Y 459.757,Z 347.363,A -85,B 0,C 180,E1 -8157.219,E2 -8157.219} C_VEL
LIN {X 0,Y 459.963,Z 342.954,A -85,B 0,C 180,E1 -8158.832,E2 -8158.832} C_VEL
LIN {X 0,Y 460.016,Z 341.258,A -85,B 0,C 180,E1 -8159.338,E2 -8159.338} C_VEL
LIN {X 0,Y 459.458,Z 338.825,A -85,B 0,C 180,E1 -8160.002,E2 -8160.002} C_VEL
LIN {X 0,Y 455.703,Z 332.654,A -85,B 0,C 180,E1 -8161.488,E2 -8161.488} C_VEL
LIN {X 0,Y 453.999,Z 328.518,A -85,B 0,C 180,E1 -8162.312,E2 -8162.312} C_VEL
LIN {X 0,Y 453.781,Z 326.177,A -85,B 0,C 180,E1 -8162.716,E2 -8162.716} C_VEL
LIN {X 0,Y 454.185,Z 318.725,A -85,B 0,C 180,E1 -8163.829,E2 -8163.829} C_VEL
LIN {X 0,Y 454.71,Z 309.458,A -85,B 0,C 180,E1 -8164.969,E2 -8164.969} C_VEL
LIN {X 0,Y 455.213,Z 298.62,A -85,B 0,C 180,E1 -8166.04,E2 -8166.04} C_VEL
LIN {X 0,Y 455.808,Z 286.714,A -85,B 0,C 180,E1 -8166.968,E2 -8166.968} C_VEL
LIN {X 0,Y 456.206,Z 274.638,A -85,B 0,C 180,E1 -8167.696,E2 -8167.696} C_VEL
LIN {X 0,Y 456.607,Z 262.194,A -85,B 0,C 180,E1 -8168.244,E2 -8168.244} C_VEL
LIN {X 0,Y 456.821,Z 249.449,A -85,B 0,C 180,E1 -8168.628,E2 -8168.628} C_VEL
LIN {X 0,Y 457.65,Z 156.518,A -85,B 0,C 180,E1 -8170.158,E2 -8170.158} C_VEL
LIN {X 0,Y 454.568,Z 141.831,A -85,B 0,C 180,E1 -8170.532,E2 -8170.532} C_VEL
LIN {X 0,Y 454.309,Z 136.277,A -85,B 0,C 180,E1 -8171.744,E2 -8171.744} C_VEL
LIN {X 0,Y 453.55,Z 131.99,A -85,B 0,C 180,E1 -8172.762,E2 -8172.762} C_VEL
LIN {X 0,Y 453.513,Z 131.997,A -85,B 0,C 180,E1 -8175.644,E2 -8175.644} C_VEL
LIN {X 0,Y 453.559,Z 131.984,A -85,B 0,C 180,E1 -8178.379,E2 -8178.379} C_VEL
LIN {X 0,Y 453.652,Z 131.974,A -85,B 0,C 180,E1 -8181.985,E2 -8181.985} C_VEL
LIN {X 0,Y 453.668,Z 131.97,A -85,B 0,C 180,E1 -8184.667,E2 -8184.667} C_VEL
LIN {X 0,Y 453.743,Z 131.967,A -85,B 0,C 180,E1 -8187.337,E2 -8187.337} C_VEL
LIN {X 0,Y 453.823,Z 131.951,A -85,B 0,C 180,E1 -8190,E2 -8190} C_VEL
LIN {X 0,Y 453.744,Z 131.961,A -85,B 0,C 180,E1 -8192.663,E2 -8192.663} C_VEL
LIN {X 0,Y 453.653,Z 131.972,A -85,B 0,C 180,E1 -8196.226,E2 -8196.226} C_VEL
LIN {X 0,Y 453.585,Z 131.985,A -85,B 0,C 180,E1 -8198.913,E2 -8198.913} C_VEL
LIN {X 0,Y 453.564,Z 131.985,A -85,B 0,C 180,E1 -8202.529,E2 -8202.529} C_VEL
LIN {X 0,Y 453.544,Z 131.986,A -85,B 0,C 180,E1 -8206.196,E2 -8206.196} C_VEL
LIN {X 0,Y 453.517,Z 131.994,A -85,B 0,C 180,E1 -8209.039,E2 -8209.039} C_VEL
LIN {X 0,Y 453.476,Z 131.994,A -85,B 0,C 180,E1 -8211.836,E2 -8211.836} C_VEL
LIN {X 0,Y 453.507,Z 131.998,A -85,B 0,C 180,E1 -8214.735,E2 -8214.735} C_VEL
LIN {X 0,Y 453.531,Z 131.988,A -85,B 0,C 180,E1 -8217.959,E2 -8217.959} C_VEL
LIN {X 0,Y 453.464,Z 131.995,A -85,B 0,C 180,E1 -8221.525,E2 -8221.525} C_VEL
LIN {X 0,Y 453.481,Z 131.997,A -85,B 0,C 180,E1 -8224.776,E2 -8224.776} C_VEL
LIN {X 0,Y 453.459,Z 132.003,A -85,B 0,C 180,E1 -8228.312,E2 -8228.312} C_VEL
LIN {X 0,Y 453.492,Z 131.996,A -85,B 0,C 180,E1 -8230.609,E2 -8230.609} C_VEL
LIN {X 0,Y 453.454,Z 131.996,A -85,B 0,C 180,E1 -8233.244,E2 -8233.244} C_VEL
LIN {X 0,Y 453.465,Z 131.998,A -85,B 0,C 180,E1 -8235.779,E2 -8235.779} C_VEL
LIN {X 0,Y 453.478,Z 132.001,A -85,B 0,C 180,E1 -8238.209,E2 -8238.209} C_VEL
LIN {X 0,Y 453.513,Z 131.99,A -85,B 0,C 180,E1 -8240.79,E2 -8240.79} C_VEL
LIN {X 0,Y 453.454,Z 132.003,A -85,B 0,C 180,E1 -8243.917,E2 -8243.917} C_VEL
LIN {X 0,Y 453.481,Z 131.993,A -85,B 0,C 180,E1 -8247.151,E2 -8247.151} C_VEL
LIN {X 0,Y 453.474,Z 131.997,A -85,B 0,C 180,E1 -8250.268,E2 -8250.268} C_VEL
LIN {X 0,Y 453.499,Z 131.993,A -85,B 0,C 180,E1 -8253.294,E2 -8253.294} C_VEL
LIN {X 0,Y 453.495,Z 131.993,A -85,B 0,C 180,E1 -8256.239,E2 -8256.239} C_VEL
LIN {X 0,Y 453.48,Z 131.995,A -85,B 0,C 180,E1 -8259.118,E2 -8259.118} C_VEL
LIN {X 0,Y 453.51,Z 131.992,A -85,B 0,C 180,E1 -8261.945,E2 -8261.945} C_VEL
LIN {X 0,Y 453.539,Z 131.986,A -85,B 0,C 180,E1 -8264.726,E2 -8264.726} C_VEL
LIN {X 0,Y 453.558,Z 131.983,A -85,B 0,C 180,E1 -8268.379,E2 -8268.379} C_VEL
LIN {X 0,Y 453.65,Z 131.973,A -85,B 0,C 180,E1 -8271.985,E2 -8271.985} C_VEL
LIN {X 0,Y 453.671,Z 131.971,A -85,B 0,C 180,E1 -8274.667,E2 -8274.667} C_VEL
LIN {X 0,Y 453.763,Z 131.964,A -85,B 0,C 180,E1 -8277.337,E2 -8277.337} C_VEL
LIN {X 0,Y 453.822,Z 131.951,A -85,B 0,C 180,E1 -8280,E2 -8280} C_VEL
LIN {X 0,Y 453.764,Z 131.961,A -85,B 0,C 180,E1 -8282.663,E2 -8282.663} C_VEL
LIN {X 0,Y 453.668,Z 131.97,A -85,B 0,C 180,E1 -8286.226,E2 -8286.226} C_VEL
LIN {X 0,Y 453.591,Z 131.987,A -85,B 0,C 180,E1 -8288.914,E2 -8288.914} C_VEL
LIN {X 0,Y 453.562,Z 131.987,A -85,B 0,C 180,E1 -8292.529,E2 -8292.529} C_VEL
LIN {X 0,Y 453.544,Z 131.987,A -85,B 0,C 180,E1 -8296.196,E2 -8296.196} C_VEL
LIN {X 0,Y 453.52,Z 131.991,A -85,B 0,C 180,E1 -8299.041,E2 -8299.041} C_VEL
LIN {X 0,Y 453.475,Z 131.994,A -85,B 0,C 180,E1 -8301.836,E2 -8301.836} C_VEL
LIN {X 0,Y 453.513,Z 131.994,A -85,B 0,C 180,E1 -8304.735,E2 -8304.735} C_VEL
LIN {X 0,Y 453.531,Z 131.989,A -85,B 0,C 180,E1 -8307.96,E2 -8307.96} C_VEL
LIN {X 0,Y 453.465,Z 131.995,A -85,B 0,C 180,E1 -8311.525,E2 -8311.525} C_VEL
LIN {X 0,Y 453.487,Z 131.994,A -85,B 0,C 180,E1 -8314.778,E2 -8314.778} C_VEL
LIN {X 0,Y 453.481,Z 131.999,A -85,B 0,C 180,E1 -8318.31,E2 -8318.31} C_VEL
LIN {X 0,Y 453.516,Z 131.991,A -85,B 0,C 180,E1 -8320.607,E2 -8320.607} C_VEL
LIN {X 0,Y 453.467,Z 132,A -85,B 0,C 180,E1 -8324.221,E2 -8324.221} C_VEL
LIN {X 0,Y 453.464,Z 131.995,A -85,B 0,C 180,E1 -8327.005,E2 -8327.005} C_VEL
LIN {X 0,Y 453.517,Z 131.991,A -85,B 0,C 180,E1 -8329.406,E2 -8329.406} C_VEL
LIN {X 0,Y 453.477,Z 131.996,A -85,B 0,C 180,E1 -8332.223,E2 -8332.223} C_VEL
LIN {X 0,Y 453.489,Z 131.994,A -85,B 0,C 180,E1 -8335.223,E2 -8335.223} C_VEL
LIN {X 0,Y 453.467,Z 131.995,A -85,B 0,C 180,E1 -8338.475,E2 -8338.475} C_VEL
LIN {X 0,Y 453.534,Z 131.993,A -85,B 0,C 180,E1 -8342.041,E2 -8342.041} C_VEL
LIN {X 0,Y 453.602,Z 132.171,A -85,B 0,C 180,E1 -8342.677,E2 -8342.677} C_VEL
LIN {X 0,Y 456.021,Z 144.197,A -85,B 0,C 180,E1 -8344.925,E2 -8344.925} C_VEL
LIN {X 0,Y 456.044,Z 149.767,A -85,B 0,C 180,E1 -8345.897,E2 -8345.897} C_VEL
LIN {X 0,Y 455.105,Z 167.771,A -85,B 0,C 180,E1 -8348.959,E2 -8348.959} C_VEL
LIN {X 0,Y 454.604,Z 181.597,A -85,B 0,C 180,E1 -8351.29,E2 -8351.29} C_VEL
LIN {X 0,Y 454.25,Z 188.737,A -85,B 0,C 180,E1 -8352.482,E2 -8352.482} C_VEL
LIN {X 0,Y 457.398,Z 211.045,A -85,B 0,C 180,E1 -8352.969,E2 -8352.969} C_VEL
LIN {X 0,Y 456.647,Z 298.241,A -85,B 0,C 180,E1 -8354.404,E2 -8354.404} C_VEL
LIN {X 0,Y 456.176,Z 311.953,A -85,B 0,C 180,E1 -8354.817,E2 -8354.817} C_VEL
LIN {X 0,Y 455.66,Z 324.33,A -85,B 0,C 180,E1 -8355.371,E2 -8355.371} C_VEL
LIN {X 0,Y 455.04,Z 337.009,A -85,B 0,C 180,E1 -8356.149,E2 -8356.149} C_VEL
LIN {X 0,Y 454.466,Z 348.408,A -85,B 0,C 180,E1 -8357.051,E2 -8357.051} C_VEL
LIN {X 0,Y 453.982,Z 358.5,A -85,B 0,C 180,E1 -8358.05,E2 -8358.05} C_VEL
LIN {X 0,Y 453.439,Z 368.508,A -85,B 0,C 180,E1 -8359.281,E2 -8359.281} C_VEL
LIN {X 0,Y 453.025,Z 377.326,A -85,B 0,C 180,E1 -8360.625,E2 -8360.625} C_VEL
LIN {X 0,Y 452.787,Z 384.36,A -85,B 0,C 180,E1 -8361.97,E2 -8361.97} C_VEL
LIN {X 0,Y 452.636,Z 390.155,A -85,B 0,C 180,E1 -8363.357,E2 -8363.357} C_VEL
LIN {X 0,Y 452.569,Z 394.41,A -85,B 0,C 180,E1 -8364.654,E2 -8364.654} C_VEL
LIN {X 0,Y 452.495,Z 396.739,A -85,B 0,C 180,E1 -8365.546,E2 -8365.546} C_VEL
LIN {X 0,Y 452.539,Z 398.638,A -85,B 0,C 180,E1 -8366.438,E2 -8366.438} C_VEL
LIN {X 0,Y 452.553,Z 400.066,A -85,B 0,C 180,E1 -8367.33,E2 -8367.33} C_VEL
LIN {X 0,Y 452.527,Z 401.073,A -85,B 0,C 180,E1 -8368.22,E2 -8368.22} C_VEL
LIN {X 0,Y 452.501,Z 401.685,A -85,B 0,C 180,E1 -8369.11,E2 -8369.11} C_VEL
LIN {X 0,Y 452.483,Z 401.902,A -85,B 0,C 180,E1 -8370,E2 -8370} C_VEL
LIN {X 0,Y 452.501,Z 401.683,A -85,B 0,C 180,E1 -8370.89,E2 -8370.89} C_VEL
LIN {X 0,Y 452.553,Z 400.042,A -85,B 0,C 180,E1 -8372.67,E2 -8372.67} C_VEL
LIN {X 0,Y 452.538,Z 398.618,A -85,B 0,C 180,E1 -8373.561,E2 -8373.561} C_VEL
LIN {X 0,Y 452.549,Z 395.626,A -85,B 0,C 180,E1 -8374.9,E2 -8374.9} C_VEL
LIN {X 0,Y 452.554,Z 391.274,A -85,B 0,C 180,E1 -8376.331,E2 -8376.331} C_VEL
LIN {X 0,Y 452.756,Z 385.377,A -85,B 0,C 180,E1 -8377.806,E2 -8377.806} C_VEL
LIN {X 0,Y 452.991,Z 378.601,A -85,B 0,C 180,E1 -8379.15,E2 -8379.15} C_VEL
LIN {X 0,Y 453.356,Z 370.211,A -85,B 0,C 180,E1 -8380.495,E2 -8380.495} C_VEL
LIN {X 0,Y 453.862,Z 361.62,A -85,B 0,C 180,E1 -8381.613,E2 -8381.613} C_VEL
LIN {X 0,Y 454.335,Z 351.568,A -85,B 0,C 180,E1 -8382.681,E2 -8382.681} C_VEL
LIN {X 0,Y 454.909,Z 340.535,A -85,B 0,C 180,E1 -8383.627,E2 -8383.627} C_VEL
LIN {X 0,Y 455.498,Z 329.056,A -85,B 0,C 180,E1 -8384.406,E2 -8384.406} C_VEL
LIN {X 0,Y 456.034,Z 317.239,A -85,B 0,C 180,E1 -8385.016,E2 -8385.016} C_VEL
LIN {X 0,Y 456.561,Z 303.68,A -85,B 0,C 180,E1 -8385.513,E2 -8385.513} C_VEL
LIN {X 0,Y 456.924,Z 290.131,A -85,B 0,C 180,E1 -8385.815,E2 -8385.815} C_VEL
LIN {X 0,Y 457.482,Z 210.334,A -85,B 0,C 180,E1 -8387.12,E2 -8387.12} C_VEL
LIN {X 0,Y 454.268,Z 187.623,A -85,B 0,C 180,E1 -8387.652,E2 -8387.652} C_VEL
LIN {X 0,Y 454.993,Z 168.666,A -85,B 0,C 180,E1 -8390.81,E2 -8390.81} C_VEL
LIN {X 0,Y 455.858,Z 150.5,A -85,B 0,C 180,E1 -8393.872,E2 -8393.872} C_VEL
LIN {X 0,Y 456.051,Z 144.893,A -85,B 0,C 180,E1 -8394.83,E2 -8394.83} C_VEL
LIN {X 0,Y 454.201,Z 134.972,A -85,B 0,C 180,E1 -8396.662,E2 -8396.662} C_VEL
LIN {X 0,Y 453.56,Z 131.989,A -85,B 0,C 180,E1 -8397.263,E2 -8397.263} C_VEL
LIN {X 0,Y 453.478,Z 131.999,A -85,B 0,C 180,E1 -8400.759,E2 -8400.759} C_VEL
LIN {X 0,Y 453.478,Z 132,A -85,B 0,C 180,E1 -8403.912,E2 -8403.912} C_VEL
LIN {X 0,Y 453.471,Z 131.999,A -85,B 0,C 180,E1 -8407.188,E2 -8407.188} C_VEL
LIN {X 0,Y 453.529,Z 131.992,A -85,B 0,C 180,E1 -8409.445,E2 -8409.445} C_VEL
LIN {X 0,Y 453.479,Z 132.002,A -85,B 0,C 180,E1 -8411.935,E2 -8411.935} C_VEL
LIN {X 0,Y 453.487,Z 131.997,A -85,B 0,C 180,E1 -8415.47,E2 -8415.47} C_VEL
LIN {X 0,Y 453.482,Z 131.998,A -85,B 0,C 180,E1 -8418.209,E2 -8418.209} C_VEL
LIN {X 0,Y 453.526,Z 131.987,A -85,B 0,C 180,E1 -8420.788,E2 -8420.788} C_VEL
LIN {X 0,Y 453.453,Z 132.001,A -85,B 0,C 180,E1 -8423.917,E2 -8423.917} C_VEL
LIN {X 0,Y 453.482,Z 131.993,A -85,B 0,C 180,E1 -8427.151,E2 -8427.151} C_VEL
LIN {X 0,Y 453.473,Z 131.993,A -85,B 0,C 180,E1 -8430.268,E2 -8430.268} C_VEL
LIN {X 0,Y 453.501,Z 131.994,A -85,B 0,C 180,E1 -8433.293,E2 -8433.293} C_VEL
LIN {X 0,Y 453.496,Z 131.991,A -85,B 0,C 180,E1 -8436.238,E2 -8436.238} C_VEL
LIN {X 0,Y 453.481,Z 131.995,A -85,B 0,C 180,E1 -8439.117,E2 -8439.117} C_VEL
LIN {X 0,Y 453.51,Z 131.991,A -85,B 0,C 180,E1 -8441.944,E2 -8441.944} C_VEL
LIN {X 0,Y 453.54,Z 131.984,A -85,B 0,C 180,E1 -8444.726,E2 -8444.726} C_VEL
LIN {X 0,Y 453.558,Z 131.981,A -85,B 0,C 180,E1 -8448.379,E2 -8448.379} C_VEL
LIN {X 0,Y 453.65,Z 131.971,A -85,B 0,C 180,E1 -8451.985,E2 -8451.985} C_VEL
LIN {X 0,Y 453.671,Z 131.972,A -85,B 0,C 180,E1 -8454.667,E2 -8454.667} C_VEL
LIN {X 0,Y 453.763,Z 131.964,A -85,B 0,C 180,E1 -8457.337,E2 -8457.337} C_VEL
LIN {X 0,Y 453.822,Z 131.949,A -85,B 0,C 180,E1 -8460,E2 -8460} C_VEL
LIN {X 0,Y 453.763,Z 131.962,A -85,B 0,C 180,E1 -8462.663,E2 -8462.663} C_VEL
LIN {X 0,Y 453.667,Z 131.969,A -85,B 0,C 180,E1 -8466.225,E2 -8466.225} C_VEL
LIN {X 0,Y 453.59,Z 131.985,A -85,B 0,C 180,E1 -8468.913,E2 -8468.913} C_VEL
LIN {X 0,Y 453.561,Z 131.988,A -85,B 0,C 180,E1 -8472.529,E2 -8472.529} C_VEL
LIN {X 0,Y 453.542,Z 131.989,A -85,B 0,C 180,E1 -8476.196,E2 -8476.196} C_VEL
LIN {X 0,Y 453.518,Z 131.993,A -85,B 0,C 180,E1 -8479.041,E2 -8479.041} C_VEL
LIN {X 0,Y 453.474,Z 131.996,A -85,B 0,C 180,E1 -8481.836,E2 -8481.836} C_VEL
LIN {X 0,Y 453.511,Z 131.999,A -85,B 0,C 180,E1 -8484.734,E2 -8484.734} C_VEL
LIN {X 0,Y 453.535,Z 131.993,A -85,B 0,C 180,E1 -8487.961,E2 -8487.961} C_VEL
LIN {X 0,Y 453.463,Z 132,A -85,B 0,C 180,E1 -8491.525,E2 -8491.525} C_VEL
LIN {X 0,Y 453.569,Z 132.092,A -85,B 0,C 180,E1 -8493.165,E2 -8493.165} C_VEL
LIN {X 0,Y 454.884,Z 139.815,A -85,B 0,C 180,E1 -8494.865,E2 -8494.865} C_VEL
LIN {X 0,Y 454.842,Z 142.66,A -85,B 0,C 180,E1 -8495.459,E2 -8495.459} C_VEL
LIN {X 0,Y 457.968,Z 156.622,A -85,B 0,C 180,E1 -8495.829,E2 -8495.829} C_VEL
LIN {X 0,Y 457.044,Z 249.677,A -85,B 0,C 180,E1 -8497.371,E2 -8497.371} C_VEL
LIN {X 0,Y 456.724,Z 263.423,A -85,B 0,C 180,E1 -8497.788,E2 -8497.788} C_VEL
LIN {X 0,Y 456.431,Z 275.263,A -85,B 0,C 180,E1 -8498.322,E2 -8498.322} C_VEL
LIN {X 0,Y 455.956,Z 287.595,A -85,B 0,C 180,E1 -8499.071,E2 -8499.071} C_VEL
LIN {X 0,Y 455.489,Z 298.591,A -85,B 0,C 180,E1 -8499.935,E2 -8499.935} C_VEL
LIN {X 0,Y 454.887,Z 309.108,A -85,B 0,C 180,E1 -8500.963,E2 -8500.963} C_VEL
LIN {X 0,Y 454.354,Z 318.148,A -85,B 0,C 180,E1 -8502.058,E2 -8502.058} C_VEL
LIN {X 0,Y 453.847,Z 326.464,A -85,B 0,C 180,E1 -8503.297,E2 -8503.297} C_VEL
LIN {X 0,Y 453.453,Z 333.196,A -85,B 0,C 180,E1 -8504.525,E2 -8504.525} C_VEL
LIN {X 0,Y 453.126,Z 339.794,A -85,B 0,C 180,E1 -8506.031,E2 -8506.031} C_VEL
LIN {X 0,Y 452.849,Z 344.821,A -85,B 0,C 180,E1 -8507.539,E2 -8507.539} C_VEL
LIN {X 0,Y 452.699,Z 347.851,A -85,B 0,C 180,E1 -8508.734,E2 -8508.734} C_VEL
LIN {X 0,Y 452.607,Z 349.433,A -85,B 0,C 180,E1 -8509.54,E2 -8509.54} C_VEL
LIN {X 0,Y 452.49,Z 351.379,A -85,B 0,C 180,E1 -8510.949,E2 -8510.949} C_VEL
LIN {X 0,Y 452.451,Z 352.37,A -85,B 0,C 180,E1 -8512.714,E2 -8512.714} C_VEL
LIN {X 0,Y 452.441,Z 352.2,A -85,B 0,C 180,E1 -8513.876,E2 -8513.876} C_VEL
LIN {X 0,Y 452.496,Z 350.92,A -85,B 0,C 180,E1 -8515.404,E2 -8515.404} C_VEL
LIN {X 0,Y 452.652,Z 348.14,A -85,B 0,C 180,E1 -8517.084,E2 -8517.084} C_VEL
LIN {X 0,Y 452.855,Z 344.316,A -85,B 0,C 180,E1 -8518.601,E2 -8518.601} C_VEL
LIN {X 0,Y 453.152,Z 338.374,A -85,B 0,C 180,E1 -8520.286,E2 -8520.286} C_VEL
LIN {X 0,Y 453.456,Z 331.932,A -85,B 0,C 180,E1 -8521.692,E2 -8521.692} C_VEL
LIN {X 0,Y 453.781,Z 326.177,A -85,B 0,C 180,E1 -8522.716,E2 -8522.716} C_VEL
LIN {X 0,Y 453.28,Z 322.578,A -85,B 0,C 180,E1 -8523.303,E2 -8523.303} C_VEL
LIN {X 0,Y 450.817,Z 316.443,A -85,B 0,C 180,E1 -8524.238,E2 -8524.238} C_VEL
LIN {X 0,Y 448.413,Z 309.812,A -85,B 0,C 180,E1 -8525.124,E2 -8525.124} C_VEL
LIN {X 0,Y 447.999,Z 305.35,A -85,B 0,C 180,E1 -8525.622,E2 -8525.622} C_VEL
LIN {X 0,Y 448.487,Z 295.045,A -85,B 0,C 180,E1 -8526.57,E2 -8526.57} C_VEL
LIN {X 0,Y 449.05,Z 283.221,A -85,B 0,C 180,E1 -8527.428,E2 -8527.428} C_VEL
LIN {X 0,Y 449.461,Z 270.419,A -85,B 0,C 180,E1 -8528.14,E2 -8528.14} C_VEL
LIN {X 0,Y 449.857,Z 257.04,A -85,B 0,C 180,E1 -8528.657,E2 -8528.657} C_VEL
LIN {X 0,Y 450.105,Z 244.032,A -85,B 0,C 180,E1 -8528.973,E2 -8528.973} C_VEL
LIN {X 0,Y 450.966,Z 157.989,A -85,B 0,C 180,E1 -8530.389,E2 -8530.389} C_VEL
LIN {X 0,Y 447.628,Z 142.148,A -85,B 0,C 180,E1 -8530.808,E2 -8530.808} C_VEL
LIN {X 0,Y 447.283,Z 137.119,A -85,B 0,C 180,E1 -8531.921,E2 -8531.921} C_VEL
LIN {X 0,Y 446.512,Z 132.867,A -85,B 0,C 180,E1 -8532.894,E2 -8532.894} C_VEL
LIN {X 0,Y 446.47,Z 132.873,A -85,B 0,C 180,E1 -8535.413,E2 -8535.413} C_VEL
LIN {X 0,Y 446.517,Z 132.862,A -85,B 0,C 180,E1 -8538.193,E2 -8538.193} C_VEL
LIN {X 0,Y 446.6,Z 132.854,A -85,B 0,C 180,E1 -8541.858,E2 -8541.858} C_VEL
LIN {X 0,Y 446.642,Z 132.845,A -85,B 0,C 180,E1 -8544.583,E2 -8544.583} C_VEL
LIN {X 0,Y 446.663,Z 132.843,A -85,B 0,C 180,E1 -8548.197,E2 -8548.197} C_VEL
LIN {X 0,Y 446.793,Z 132.827,A -85,B 0,C 180,E1 -8550,E2 -8550} C_VEL
LIN {X 0,Y 446.691,Z 132.84,A -85,B 0,C 180,E1 -8552.705,E2 -8552.705} C_VEL
LIN {X 0,Y 446.621,Z 132.848,A -85,B 0,C 180,E1 -8556.324,E2 -8556.324} C_VEL
LIN {X 0,Y 446.521,Z 132.86,A -85,B 0,C 180,E1 -8559.97,E2 -8559.97} C_VEL
LIN {X 0,Y 446.521,Z 132.864,A -85,B 0,C 180,E1 -8562.73,E2 -8562.73} C_VEL
LIN {X 0,Y 446.495,Z 132.864,A -85,B 0,C 180,E1 -8566.227,E2 -8566.227} C_VEL
LIN {X 0,Y 446.468,Z 132.869,A -85,B 0,C 180,E1 -8569.303,E2 -8569.303} C_VEL
LIN {X 0,Y 446.418,Z 132.874,A -85,B 0,C 180,E1 -8572.199,E2 -8572.199} C_VEL
LIN {X 0,Y 446.449,Z 132.872,A -85,B 0,C 180,E1 -8575.153,E2 -8575.153} C_VEL
LIN {X 0,Y 446.484,Z 132.867,A -85,B 0,C 180,E1 -8578.179,E2 -8578.179} C_VEL
LIN {X 0,Y 446.417,Z 132.873,A -85,B 0,C 180,E1 -8581.775,E2 -8581.775} C_VEL
LIN {X 0,Y 446.422,Z 132.88,A -85,B 0,C 180,E1 -8584.523,E2 -8584.523} C_VEL
LIN {X 0,Y 446.412,Z 132.877,A -85,B 0,C 180,E1 -8588.079,E2 -8588.079} C_VEL
LIN {X 0,Y 446.425,Z 132.873,A -85,B 0,C 180,E1 -8590.917,E2 -8590.917} C_VEL
LIN {X 0,Y 446.4,Z 132.878,A -85,B 0,C 180,E1 -8593.846,E2 -8593.846} C_VEL
LIN {X 0,Y 446.398,Z 132.88,A -85,B 0,C 180,E1 -8596.403,E2 -8596.403} C_VEL
LIN {X 0,Y 446.425,Z 132.872,A -85,B 0,C 180,E1 -8599.082,E2 -8599.082} C_VEL
LIN {X 0,Y 446.429,Z 132.878,A -85,B 0,C 180,E1 -8601.918,E2 -8601.918} C_VEL
LIN {X 0,Y 446.428,Z 132.874,A -85,B 0,C 180,E1 -8605.477,E2 -8605.477} C_VEL
LIN {X 0,Y 446.414,Z 132.874,A -85,B 0,C 180,E1 -8608.7,E2 -8608.7} C_VEL
LIN {X 0,Y 446.483,Z 132.873,A -85,B 0,C 180,E1 -8611.821,E2 -8611.821} C_VEL
LIN {X 0,Y 446.442,Z 132.87,A -85,B 0,C 180,E1 -8614.847,E2 -8614.847} C_VEL
LIN {X 0,Y 446.446,Z 132.871,A -85,B 0,C 180,E1 -8618.245,E2 -8618.245} C_VEL
LIN {X 0,Y 446.456,Z 132.875,A -85,B 0,C 180,E1 -8621.649,E2 -8621.649} C_VEL
LIN {X 0,Y 446.507,Z 132.862,A -85,B 0,C 180,E1 -8624.48,E2 -8624.48} C_VEL
LIN {X 0,Y 446.516,Z 132.861,A -85,B 0,C 180,E1 -8628.193,E2 -8628.193} C_VEL
LIN {X 0,Y 446.599,Z 132.852,A -85,B 0,C 180,E1 -8631.858,E2 -8631.858} C_VEL
LIN {X 0,Y 446.645,Z 132.846,A -85,B 0,C 180,E1 -8634.583,E2 -8634.583} C_VEL
LIN {X 0,Y 446.707,Z 132.843,A -85,B 0,C 180,E1 -8637.295,E2 -8637.295} C_VEL
LIN {X 0,Y 446.793,Z 132.826,A -85,B 0,C 180,E1 -8640,E2 -8640} C_VEL
LIN {X 0,Y 446.707,Z 132.84,A -85,B 0,C 180,E1 -8642.705,E2 -8642.705} C_VEL
LIN {X 0,Y 446.638,Z 132.847,A -85,B 0,C 180,E1 -8646.324,E2 -8646.324} C_VEL
LIN {X 0,Y 446.537,Z 132.864,A -85,B 0,C 180,E1 -8649.056,E2 -8649.056} C_VEL
LIN {X 0,Y 446.52,Z 132.867,A -85,B 0,C 180,E1 -8652.73,E2 -8652.73} C_VEL
LIN {X 0,Y 446.495,Z 132.866,A -85,B 0,C 180,E1 -8656.228,E2 -8656.228} C_VEL
LIN {X 0,Y 446.469,Z 132.867,A -85,B 0,C 180,E1 -8659.303,E2 -8659.303} C_VEL
LIN {X 0,Y 446.417,Z 132.876,A -85,B 0,C 180,E1 -8662.2,E2 -8662.2} C_VEL
LIN {X 0,Y 446.456,Z 132.869,A -85,B 0,C 180,E1 -8665.153,E2 -8665.153} C_VEL
LIN {X 0,Y 446.484,Z 132.87,A -85,B 0,C 180,E1 -8668.179,E2 -8668.179} C_VEL
LIN {X 0,Y 446.418,Z 132.875,A -85,B 0,C 180,E1 -8671.775,E2 -8671.775} C_VEL
LIN {X 0,Y 446.429,Z 132.876,A -85,B 0,C 180,E1 -8674.523,E2 -8674.523} C_VEL
LIN {X 0,Y 446.435,Z 132.878,A -85,B 0,C 180,E1 -8678.083,E2 -8678.083} C_VEL
LIN {X 0,Y 446.443,Z 132.87,A -85,B 0,C 180,E1 -8680.92,E2 -8680.92} C_VEL
LIN {X 0,Y 446.402,Z 132.881,A -85,B 0,C 180,E1 -8683.846,E2 -8683.846} C_VEL
LIN {X 0,Y 446.4,Z 132.878,A -85,B 0,C 180,E1 -8686.404,E2 -8686.404} C_VEL
LIN {X 0,Y 446.469,Z 132.874,A -85,B 0,C 180,E1 -8689.805,E2 -8689.805} C_VEL
LIN {X 0,Y 446.433,Z 132.875,A -85,B 0,C 180,E1 -8692.124,E2 -8692.124} C_VEL
LIN {X 0,Y 446.431,Z 132.876,A -85,B 0,C 180,E1 -8695.477,E2 -8695.477} C_VEL
LIN {X 0,Y 446.417,Z 132.874,A -85,B 0,C 180,E1 -8698.7,E2 -8698.7} C_VEL
LIN {X 0,Y 446.519,Z 132.865,A -85,B 0,C 180,E1 -8702.334,E2 -8702.334} C_VEL
LIN {X 0,Y 446.574,Z 133.102,A -85,B 0,C 180,E1 -8702.465,E2 -8702.465} C_VEL
LIN {X 0,Y 449.214,Z 146.539,A -85,B 0,C 180,E1 -8705.013,E2 -8705.013} C_VEL
LIN {X 0,Y 448.606,Z 158.858,A -85,B 0,C 180,E1 -8707.157,E2 -8707.157} C_VEL
LIN {X 0,Y 447.878,Z 177.155,A -85,B 0,C 180,E1 -8710.307,E2 -8710.307} C_VEL
LIN {X 0,Y 447.253,Z 188.325,A -85,B 0,C 180,E1 -8712.204,E2 -8712.204} C_VEL
LIN {X 0,Y 450.592,Z 212.376,A -85,B 0,C 180,E1 -8712.746,E2 -8712.746} C_VEL
LIN {X 0,Y 449.78,Z 297.257,A -85,B 0,C 180,E1 -8714.16,E2 -8714.16} C_VEL
LIN {X 0,Y 449.363,Z 310.412,A -85,B 0,C 180,E1 -8714.552,E2 -8714.552} C_VEL
LIN {X 0,Y 448.815,Z 322.547,A -85,B 0,C 180,E1 -8715.085,E2 -8715.085} C_VEL
LIN {X 0,Y 448.22,Z 334.835,A -85,B 0,C 180,E1 -8715.818,E2 -8715.818} C_VEL
LIN {X 0,Y 447.606,Z 346.331,A -85,B 0,C 180,E1 -8716.712,E2 -8716.712} C_VEL
LIN {X 0,Y 447.03,Z 356.954,A -85,B 0,C 180,E1 -8717.746,E2 -8717.746} C_VEL
LIN {X 0,Y 446.556,Z 366.39,A -85,B 0,C 180,E1 -8718.884,E2 -8718.884} C_VEL
LIN {X 0,Y 446.055,Z 375.506,A -85,B 0,C 180,E1 -8720.249,E2 -8720.249} C_VEL
LIN {X 0,Y 445.765,Z 382.856,A -85,B 0,C 180,E1 -8721.614,E2 -8721.614} C_VEL
LIN {X 0,Y 445.594,Z 387.824,A -85,B 0,C 180,E1 -8722.751,E2 -8722.751} C_VEL
LIN {X 0,Y 445.451,Z 392.215,A -85,B 0,C 180,E1 -8723.979,E2 -8723.979} C_VEL
LIN {X 0,Y 445.42,Z 396.33,A -85,B 0,C 180,E1 -8725.475,E2 -8725.475} C_VEL
LIN {X 0,Y 445.437,Z 398.233,A -85,B 0,C 180,E1 -8726.382,E2 -8726.382} C_VEL
LIN {X 0,Y 445.476,Z 399.669,A -85,B 0,C 180,E1 -8727.287,E2 -8727.287} C_VEL
LIN {X 0,Y 445.437,Z 401.294,A -85,B 0,C 180,E1 -8729.096,E2 -8729.096} C_VEL
LIN {X 0,Y 445.418,Z 401.514,A -85,B 0,C 180,E1 -8730,E2 -8730} C_VEL
LIN {X 0,Y 445.437,Z 401.299,A -85,B 0,C 180,E1 -8730.904,E2 -8730.904} C_VEL
LIN {X 0,Y 445.476,Z 399.659,A -85,B 0,C 180,E1 -8732.713,E2 -8732.713} C_VEL
LIN {X 0,Y 445.436,Z 398.235,A -85,B 0,C 180,E1 -8733.618,E2 -8733.618} C_VEL
LIN {X 0,Y 445.478,Z 395.247,A -85,B 0,C 180,E1 -8734.978,E2 -8734.978} C_VEL
LIN {X 0,Y 445.456,Z 391.204,A -85,B 0,C 180,E1 -8736.341,E2 -8736.341} C_VEL
LIN {X 0,Y 445.697,Z 385.008,A -85,B 0,C 180,E1 -8737.931,E2 -8737.931} C_VEL
LIN {X 0,Y 445.925,Z 378.238,A -85,B 0,C 180,E1 -8739.296,E2 -8739.296} C_VEL
LIN {X 0,Y 446.32,Z 369.851,A -85,B 0,C 180,E1 -8740.662,E2 -8740.662} C_VEL
LIN {X 0,Y 446.865,Z 361.269,A -85,B 0,C 180,E1 -8741.798,E2 -8741.798} C_VEL
LIN {X 0,Y 447.358,Z 351.666,A -85,B 0,C 180,E1 -8742.84,E2 -8742.84} C_VEL
LIN {X 0,Y 447.98,Z 340.216,A -85,B 0,C 180,E1 -8743.842,E2 -8743.842} C_VEL
LIN {X 0,Y 448.625,Z 328.769,A -85,B 0,C 180,E1 -8744.632,E2 -8744.632} C_VEL
LIN {X 0,Y 449.179,Z 317.016,A -85,B 0,C 180,E1 -8745.251,E2 -8745.251} C_VEL
LIN {X 0,Y 449.728,Z 303.549,A -85,B 0,C 180,E1 -8745.755,E2 -8745.755} C_VEL
LIN {X 0,Y 450.099,Z 290.293,A -85,B 0,C 180,E1 -8746.061,E2 -8746.061} C_VEL
LIN {X 0,Y 450.712,Z 211.186,A -85,B 0,C 180,E1 -8747.376,E2 -8747.376} C_VEL
LIN {X 0,Y 447.302,Z 187.185,A -85,B 0,C 180,E1 -8747.953,E2 -8747.953} C_VEL
LIN {X 0,Y 448.081,Z 168.344,A -85,B 0,C 180,E1 -8751.146,E2 -8751.146} C_VEL
LIN {X 0,Y 449.099,Z 149.127,A -85,B 0,C 180,E1 -8754.438,E2 -8754.438} C_VEL
LIN {X 0,Y 448.882,Z 144.563,A -85,B 0,C 180,E1 -8755.255,E2 -8755.255} C_VEL
LIN {X 0,Y 446.518,Z 132.867,A -85,B 0,C 180,E1 -8757.507,E2 -8757.507} C_VEL
LIN {X 0,Y 446.429,Z 132.879,A -85,B 0,C 180,E1 -8760.249,E2 -8760.249} C_VEL
LIN {X 0,Y 446.446,Z 132.873,A -85,B 0,C 180,E1 -8763.453,E2 -8763.453} C_VEL
LIN {X 0,Y 446.409,Z 132.88,A -85,B 0,C 180,E1 -8766.744,E2 -8766.744} C_VEL
LIN {X 0,Y 446.489,Z 132.869,A -85,B 0,C 180,E1 -8769.53,E2 -8769.53} C_VEL
LIN {X 0,Y 446.43,Z 132.877,A -85,B 0,C 180,E1 -8772.604,E2 -8772.604} C_VEL
LIN {X 0,Y 446.454,Z 132.872,A -85,B 0,C 180,E1 -8775.103,E2 -8775.103} C_VEL
LIN {X 0,Y 446.435,Z 132.873,A -85,B 0,C 180,E1 -8778.609,E2 -8778.609} C_VEL
LIN {X 0,Y 446.47,Z 132.866,A -85,B 0,C 180,E1 -8780.975,E2 -8780.975} C_VEL
LIN {X 0,Y 446.418,Z 132.875,A -85,B 0,C 180,E1 -8784.374,E2 -8784.374} C_VEL
LIN {X 0,Y 446.421,Z 132.876,A -85,B 0,C 180,E1 -8787.638,E2 -8787.638} C_VEL
LIN {X 0,Y 446.447,Z 132.867,A -85,B 0,C 180,E1 -8790.79,E2 -8790.79} C_VEL
LIN {X 0,Y 446.477,Z 132.867,A -85,B 0,C 180,E1 -8793.848,E2 -8793.848} C_VEL
LIN {X 0,Y 446.424,Z 132.871,A -85,B 0,C 180,E1 -8796.823,E2 -8796.823} C_VEL
LIN {X 0,Y 446.443,Z 132.872,A -85,B 0,C 180,E1 -8799.737,E2 -8799.737} C_VEL
LIN {X 0,Y 446.462,Z 132.867,A -85,B 0,C 180,E1 -8802.597,E2 -8802.597} C_VEL
LIN {X 0,Y 446.47,Z 132.869,A -85,B 0,C 180,E1 -8805.412,E2 -8805.412} C_VEL
LIN {X 0,Y 446.516,Z 132.859,A -85,B 0,C 180,E1 -8808.193,E2 -8808.193} C_VEL
LIN {X 0,Y 446.599,Z 132.85,A -85,B 0,C 180,E1 -8811.858,E2 -8811.858} C_VEL
LIN {X 0,Y 446.645,Z 132.847,A -85,B 0,C 180,E1 -8814.582,E2 -8814.582} C_VEL
LIN {X 0,Y 446.706,Z 132.844,A -85,B 0,C 180,E1 -8817.295,E2 -8817.295} C_VEL
LIN {X 0,Y 446.792,Z 132.825,A -85,B 0,C 180,E1 -8820,E2 -8820} C_VEL
LIN {X 0,Y 446.707,Z 132.842,A -85,B 0,C 180,E1 -8822.705,E2 -8822.705} C_VEL
LIN {X 0,Y 446.637,Z 132.846,A -85,B 0,C 180,E1 -8826.324,E2 -8826.324} C_VEL
LIN {X 0,Y 446.536,Z 132.864,A -85,B 0,C 180,E1 -8829.055,E2 -8829.055} C_VEL
LIN {X 0,Y 446.519,Z 132.868,A -85,B 0,C 180,E1 -8832.73,E2 -8832.73} C_VEL
LIN {X 0,Y 446.494,Z 132.867,A -85,B 0,C 180,E1 -8836.228,E2 -8836.228} C_VEL
LIN {X 0,Y 446.467,Z 132.869,A -85,B 0,C 180,E1 -8839.303,E2 -8839.303} C_VEL
LIN {X 0,Y 446.416,Z 132.879,A -85,B 0,C 180,E1 -8842.2,E2 -8842.2} C_VEL
LIN {X 0,Y 446.455,Z 132.875,A -85,B 0,C 180,E1 -8845.152,E2 -8845.152} C_VEL
LIN {X 0,Y 446.482,Z 132.871,A -85,B 0,C 180,E1 -8848.179,E2 -8848.179} C_VEL
LIN {X 0,Y 446.414,Z 132.878,A -85,B 0,C 180,E1 -8851.3,E2 -8851.3} C_VEL
LIN {X 0,Y 446.489,Z 132.955,A -85,B 0,C 180,E1 -8852.925,E2 -8852.925} C_VEL
LIN {X 0,Y 447.927,Z 140.697,A -85,B 0,C 180,E1 -8854.664,E2 -8854.664} C_VEL
LIN {X 0,Y 447.931,Z 142.957,A -85,B 0,C 180,E1 -8855.147,E2 -8855.147} C_VEL
LIN {X 0,Y 451.266,Z 157.742,A -85,B 0,C 180,E1 -8855.562,E2 -8855.562} C_VEL
LIN {X 0,Y 450.261,Z 250.251,A -85,B 0,C 180,E1 -8857.124,E2 -8857.124} C_VEL
LIN {X 0,Y 449.937,Z 263.477,A -85,B 0,C 180,E1 -8857.53,E2 -8857.53} C_VEL
LIN {X 0,Y 449.598,Z 275.192,A -85,B 0,C 180,E1 -8858.059,E2 -8858.059} C_VEL
LIN {X 0,Y 449.148,Z 286.651,A -85,B 0,C 180,E1 -8858.748,E2 -8858.748} C_VEL
LIN {X 0,Y 448.657,Z 297.693,A -85,B 0,C 180,E1 -8859.606,E2 -8859.606} C_VEL
LIN {X 0,Y 448.037,Z 308.114,A -85,B 0,C 180,E1 -8860.615,E2 -8860.615} C_VEL
LIN {X 0,Y 447.463,Z 317.615,A -85,B 0,C 180,E1 -8861.751,E2 -8861.751} C_VEL
LIN {X 0,Y 446.921,Z 326.125,A -85,B 0,C 180,E1 -8863.011,E2 -8863.011} C_VEL
LIN {X 0,Y 446.45,Z 333.439,A -85,B 0,C 180,E1 -8864.351,E2 -8864.351} C_VEL
LIN {X 0,Y 446.136,Z 339.038,A -85,B 0,C 180,E1 -8865.619,E2 -8865.619} C_VEL
LIN {X 0,Y 445.902,Z 343.562,A -85,B 0,C 180,E1 -8866.893,E2 -8866.893} C_VEL
LIN {X 0,Y 445.652,Z 347.932,A -85,B 0,C 180,E1 -8868.521,E2 -8868.521} C_VEL
LIN {X 0,Y 445.505,Z 350.181,A -85,B 0,C 180,E1 -8869.7,E2 -8869.7} C_VEL
LIN {X 0,Y 445.413,Z 351.733,A -85,B 0,C 180,E1 -8870.866,E2 -8870.866} C_VEL
LIN {X 0,Y 445.386,Z 352.597,A -85,B 0,C 180,E1 -8872.09,E2 -8872.09} C_VEL
LIN {X 0,Y 445.343,Z 352.693,A -85,B 0,C 180,E1 -8873.594,E2 -8873.594} C_VEL
LIN {X 0,Y 445.421,Z 351.358,A -85,B 0,C 180,E1 -8875.388,E2 -8875.388} C_VEL
LIN {X 0,Y 445.52,Z 349.338,A -85,B 0,C 180,E1 -8876.727,E2 -8876.727} C_VEL
LIN {X 0,Y 445.747,Z 345.558,A -85,B 0,C 180,E1 -8878.365,E2 -8878.365} C_VEL
LIN {X 0,Y 446.04,Z 340.036,A -85,B 0,C 180,E1 -8880.066,E2 -8880.066} C_VEL
LIN {X 0,Y 446.335,Z 333.594,A -85,B 0,C 180,E1 -8881.555,E2 -8881.555} C_VEL
LIN {X 0,Y 446.766,Z 326.53,A -85,B 0,C 180,E1 -8882.858,E2 -8882.858} C_VEL
LIN {X 0,Y 447.279,Z 317.917,A -85,B 0,C 180,E1 -8884.149,E2 -8884.149} C_VEL
LIN {X 0,Y 447.805,Z 308.747,A -85,B 0,C 180,E1 -8885.263,E2 -8885.263} C_VEL
LIN {X 0,Y 447.999,Z 305.35,A -85,B 0,C 180,E1 -8885.622,E2 -8885.622} C_VEL
LIN {X 0,Y 447.557,Z 300.781,A -85,B 0,C 180,E1 -8886.102,E2 -8886.102} C_VEL
LIN {X 0,Y 445.065,Z 293.154,A -85,B 0,C 180,E1 -8886.859,E2 -8886.859} C_VEL
LIN {X 0,Y 442.639,Z 285.084,A -85,B 0,C 180,E1 -8887.532,E2 -8887.532} C_VEL
LIN {X 0,Y 442.288,Z 279.827,A -85,B 0,C 180,E1 -8887.875,E2 -8887.875} C_VEL
LIN {X 0,Y 442.734,Z 267.105,A -85,B 0,C 180,E1 -8888.525,E2 -8888.525} C_VEL
LIN {X 0,Y 443.073,Z 255.067,A -85,B 0,C 180,E1 -8888.96,E2 -8888.96} C_VEL
LIN {X 0,Y 443.262,Z 241.793,A -85,B 0,C 180,E1 -8889.254,E2 -8889.254} C_VEL
LIN {X 0,Y 444.076,Z 158.565,A -85,B 0,C 180,E1 -8890.649,E2 -8890.649} C_VEL
LIN {X 0,Y 440.67,Z 142.548,A -85,B 0,C 180,E1 -8891.068,E2 -8891.068} C_VEL
LIN {X 0,Y 440.069,Z 136.931,A -85,B 0,C 180,E1 -8892.336,E2 -8892.336} C_VEL
LIN {X 0,Y 439.455,Z 133.747,A -85,B 0,C 180,E1 -8893.09,E2 -8893.09} C_VEL
LIN {X 0,Y 439.423,Z 133.75,A -85,B 0,C 180,E1 -8896.119,E2 -8896.119} C_VEL
LIN {X 0,Y 439.435,Z 133.744,A -85,B 0,C 180,E1 -8898.935,E2 -8898.935} C_VEL
LIN {X 0,Y 439.599,Z 133.722,A -85,B 0,C 180,E1 -8902.397,E2 -8902.397} C_VEL
LIN {X 0,Y 439.618,Z 133.72,A -85,B 0,C 180,E1 -8904.496,E2 -8904.496} C_VEL
LIN {X 0,Y 439.633,Z 133.719,A -85,B 0,C 180,E1 -8908.168,E2 -8908.168} C_VEL
LIN {X 0,Y 439.763,Z 133.703,A -85,B 0,C 180,E1 -8910,E2 -8910} C_VEL
LIN {X 0,Y 439.64,Z 133.719,A -85,B 0,C 180,E1 -8912.749,E2 -8912.749} C_VEL
LIN {X 0,Y 439.593,Z 133.724,A -85,B 0,C 180,E1 -8916.426,E2 -8916.426} C_VEL
LIN {X 0,Y 439.496,Z 133.742,A -85,B 0,C 180,E1 -8919.202,E2 -8919.202} C_VEL
LIN {X 0,Y 439.466,Z 133.746,A -85,B 0,C 180,E1 -8922.938,E2 -8922.938} C_VEL
LIN {X 0,Y 439.446,Z 133.743,A -85,B 0,C 180,E1 -8926.348,E2 -8926.348} C_VEL
LIN {X 0,Y 439.402,Z 133.747,A -85,B 0,C 180,E1 -8929.626,E2 -8929.626} C_VEL
LIN {X 0,Y 439.364,Z 133.757,A -85,B 0,C 180,E1 -8932.575,E2 -8932.575} C_VEL
LIN {X 0,Y 439.4,Z 133.747,A -85,B 0,C 180,E1 -8935.585,E2 -8935.585} C_VEL
LIN {X 0,Y 439.416,Z 133.752,A -85,B 0,C 180,E1 -8938.673,E2 -8938.673} C_VEL
LIN {X 0,Y 439.367,Z 133.753,A -85,B 0,C 180,E1 -8942.03,E2 -8942.03} C_VEL
LIN {X 0,Y 439.391,Z 133.748,A -85,B 0,C 180,E1 -8945.34,E2 -8945.34} C_VEL
LIN {X 0,Y 439.374,Z 133.755,A -85,B 0,C 180,E1 -8948.596,E2 -8948.596} C_VEL
LIN {X 0,Y 439.387,Z 133.749,A -85,B 0,C 180,E1 -8951.257,E2 -8951.257} C_VEL
LIN {X 0,Y 439.4,Z 133.749,A -85,B 0,C 180,E1 -8954.729,E2 -8954.729} C_VEL
LIN {X 0,Y 439.394,Z 133.751,A -85,B 0,C 180,E1 -8957.796,E2 -8957.796} C_VEL
LIN {X 0,Y 439.435,Z 133.749,A -85,B 0,C 180,E1 -8960.228,E2 -8960.228} C_VEL
LIN {X 0,Y 439.375,Z 133.754,A -85,B 0,C 180,E1 -8963.713,E2 -8963.713} C_VEL
LIN {X 0,Y 439.37,Z 133.751,A -85,B 0,C 180,E1 -8967.054,E2 -8967.054} C_VEL
LIN {X 0,Y 439.381,Z 133.752,A -85,B 0,C 180,E1 -8970.274,E2 -8970.274} C_VEL
LIN {X 0,Y 439.426,Z 133.747,A -85,B 0,C 180,E1 -8973.396,E2 -8973.396} C_VEL
LIN {X 0,Y 439.381,Z 133.75,A -85,B 0,C 180,E1 -8976.429,E2 -8976.429} C_VEL
LIN {X 0,Y 439.386,Z 133.754,A -85,B 0,C 180,E1 -8979.397,E2 -8979.397} C_VEL
LIN {X 0,Y 439.43,Z 133.744,A -85,B 0,C 180,E1 -8982.31,E2 -8982.31} C_VEL
LIN {X 0,Y 439.447,Z 133.745,A -85,B 0,C 180,E1 -8985.174,E2 -8985.174} C_VEL
LIN {X 0,Y 439.482,Z 133.738,A -85,B 0,C 180,E1 -8988.001,E2 -8988.001} C_VEL
LIN {X 0,Y 439.546,Z 133.732,A -85,B 0,C 180,E1 -8991.726,E2 -8991.726} C_VEL
LIN {X 0,Y 439.621,Z 133.72,A -85,B 0,C 180,E1 -8994.496,E2 -8994.496} C_VEL
LIN {X 0,Y 439.634,Z 133.718,A -85,B 0,C 180,E1 -8998.168,E2 -8998.168} C_VEL
LIN {X 0,Y 439.762,Z 133.702,A -85,B 0,C 180,E1 -9000,E2 -9000} C_VEL
LIN {X 0,Y 439.654,Z 133.72,A -85,B 0,C 180,E1 -9002.749,E2 -9002.749} C_VEL
LIN {X 0,Y 439.61,Z 133.723,A -85,B 0,C 180,E1 -9006.426,E2 -9006.426} C_VEL
LIN {X 0,Y 439.499,Z 133.738,A -85,B 0,C 180,E1 -9009.202,E2 -9009.202} C_VEL
LIN {X 0,Y 439.464,Z 133.745,A -85,B 0,C 180,E1 -9012.938,E2 -9012.938} C_VEL
LIN {X 0,Y 439.446,Z 133.745,A -85,B 0,C 180,E1 -9016.349,E2 -9016.349} C_VEL
LIN {X 0,Y 439.402,Z 133.747,A -85,B 0,C 180,E1 -9019.627,E2 -9019.627} C_VEL
LIN {X 0,Y 439.364,Z 133.759,A -85,B 0,C 180,E1 -9022.576,E2 -9022.576} C_VEL
LIN {X 0,Y 439.404,Z 133.747,A -85,B 0,C 180,E1 -9025.585,E2 -9025.585} C_VEL
LIN {X 0,Y 439.417,Z 133.749,A -85,B 0,C 180,E1 -9028.674,E2 -9028.674} C_VEL
LIN {X 0,Y 439.369,Z 133.755,A -85,B 0,C 180,E1 -9032.031,E2 -9032.031} C_VEL
LIN {X 0,Y 439.394,Z 133.748,A -85,B 0,C 180,E1 -9035.341,E2 -9035.341} C_VEL
LIN {X 0,Y 439.396,Z 133.75,A -85,B 0,C 180,E1 -9038.594,E2 -9038.594} C_VEL
LIN {X 0,Y 439.399,Z 133.748,A -85,B 0,C 180,E1 -9041.259,E2 -9041.259} C_VEL
LIN {X 0,Y 439.402,Z 133.747,A -85,B 0,C 180,E1 -9044.73,E2 -9044.73} C_VEL
LIN {X 0,Y 439.398,Z 133.754,A -85,B 0,C 180,E1 -9047.796,E2 -9047.796} C_VEL
LIN {X 0,Y 439.45,Z 133.744,A -85,B 0,C 180,E1 -9050.23,E2 -9050.23} C_VEL
LIN {X 0,Y 439.377,Z 133.757,A -85,B 0,C 180,E1 -9053.713,E2 -9053.713} C_VEL
LIN {X 0,Y 439.374,Z 133.752,A -85,B 0,C 180,E1 -9057.054,E2 -9057.054} C_VEL
LIN {X 0,Y 439.384,Z 133.754,A -85,B 0,C 180,E1 -9060.274,E2 -9060.274} C_VEL
LIN {X 0,Y 439.465,Z 133.754,A -85,B 0,C 180,E1 -9062.192,E2 -9062.192} C_VEL
LIN {X 0,Y 442.287,Z 147.906,A -85,B 0,C 180,E1 -9064.923,E2 -9064.923} C_VEL
LIN {X 0,Y 441.526,Z 164.116,A -85,B 0,C 180,E1 -9067.788,E2 -9067.788} C_VEL
LIN {X 0,Y 440.57,Z 183.466,A -85,B 0,C 180,E1 -9071.154,E2 -9071.154} C_VEL
LIN {X 0,Y 440.302,Z 188.11,A -85,B 0,C 180,E1 -9071.938,E2 -9071.938} C_VEL
LIN {X 0,Y 443.799,Z 213.669,A -85,B 0,C 180,E1 -9072.514,E2 -9072.514} C_VEL
LIN {X 0,Y 442.899,Z 297.384,A -85,B 0,C 180,E1 -9073.937,E2 -9073.937} C_VEL
LIN {X 0,Y 442.455,Z 311.132,A -85,B 0,C 180,E1 -9074.364,E2 -9074.364} C_VEL
LIN {X 0,Y 441.885,Z 322.987,A -85,B 0,C 180,E1 -9074.904,E2 -9074.904} C_VEL
LIN {X 0,Y 441.3,Z 334.238,A -85,B 0,C 180,E1 -9075.591,E2 -9075.591} C_VEL
LIN {X 0,Y 440.666,Z 345.569,A -85,B 0,C 180,E1 -9076.481,E2 -9076.481} C_VEL
LIN {X 0,Y 440.006,Z 356.424,A -85,B 0,C 180,E1 -9077.548,E2 -9077.548} C_VEL
LIN {X 0,Y 439.537,Z 365.899,A -85,B 0,C 180,E1 -9078.704,E2 -9078.704} C_VEL
LIN {X 0,Y 438.98,Z 375.032,A -85,B 0,C 180,E1 -9080.09,E2 -9080.09} C_VEL
LIN {X 0,Y 438.69,Z 382.401,A -85,B 0,C 180,E1 -9081.478,E2 -9081.478} C_VEL
LIN {X 0,Y 438.516,Z 387.384,A -85,B 0,C 180,E1 -9082.634,E2 -9082.634} C_VEL
LIN {X 0,Y 438.353,Z 392.214,A -85,B 0,C 180,E1 -9084.018,E2 -9084.018} C_VEL
LIN {X 0,Y 438.348,Z 395.917,A -85,B 0,C 180,E1 -9085.402,E2 -9085.402} C_VEL
LIN {X 0,Y 438.338,Z 397.823,A -85,B 0,C 180,E1 -9086.323,E2 -9086.323} C_VEL
LIN {X 0,Y 438.401,Z 399.269,A -85,B 0,C 180,E1 -9087.243,E2 -9087.243} C_VEL
LIN {X 0,Y 438.375,Z 400.902,A -85,B 0,C 180,E1 -9089.081,E2 -9089.081} C_VEL
LIN {X 0,Y 438.355,Z 401.126,A -85,B 0,C 180,E1 -9090,E2 -9090} C_VEL
LIN {X 0,Y 438.359,Z 400.915,A -85,B 0,C 180,E1 -9090.919,E2 -9090.919} C_VEL
LIN {X 0,Y 438.401,Z 399.28,A -85,B 0,C 180,E1 -9092.757,E2 -9092.757} C_VEL
LIN {X 0,Y 438.336,Z 397.857,A -85,B 0,C 180,E1 -9093.677,E2 -9093.677} C_VEL
LIN {X 0,Y 438.406,Z 394.872,A -85,B 0,C 180,E1 -9095.058,E2 -9095.058} C_VEL
LIN {X 0,Y 438.369,Z 390.831,A -85,B 0,C 180,E1 -9096.444,E2 -9096.444} C_VEL
LIN {X 0,Y 438.623,Z 384.642,A -85,B 0,C 180,E1 -9098.059,E2 -9098.059} C_VEL
LIN {X 0,Y 438.865,Z 377.878,A -85,B 0,C 180,E1 -9099.447,E2 -9099.447} C_VEL
LIN {X 0,Y 439.314,Z 369.503,A -85,B 0,C 180,E1 -9100.834,E2 -9100.834} C_VEL
LIN {X 0,Y 439.875,Z 360.937,A -85,B 0,C 180,E1 -9101.988,E2 -9101.988} C_VEL
LIN {X 0,Y 440.438,Z 350.908,A -85,B 0,C 180,E1 -9103.089,E2 -9103.089} C_VEL
LIN {X 0,Y 441.064,Z 339.922,A -85,B 0,C 180,E1 -9104.063,E2 -9104.063} C_VEL
LIN {X 0,Y 441.752,Z 328.503,A -85,B 0,C 180,E1 -9104.865,E2 -9104.865} C_VEL
LIN {X 0,Y 442.338,Z 316.819,A -85,B 0,C 180,E1 -9105.493,E2 -9105.493} C_VEL
LIN {X 0,Y 442.909,Z 303.462,A -85,B 0,C 180,E1 -9106.004,E2 -9106.004} C_VEL
LIN {X 0,Y 443.303,Z 290.49,A -85,B 0,C 180,E1 -9106.314,E2 -9106.314} C_VEL
LIN {X 0,Y 444.054,Z 212.564,A -85,B 0,C 180,E1 -9107.631,E2 -9107.631} C_VEL
LIN {X 0,Y 440.545,Z 188.357,A -85,B 0,C 180,E1 -9108.209,E2 -9108.209} C_VEL
LIN {X 0,Y 440.342,Z 186.785,A -85,B 0,C 180,E1 -9108.261,E2 -9108.261} C_VEL
LIN {X 0,Y 441.215,Z 168.021,A -85,B 0,C 180,E1 -9111.491,E2 -9111.491} C_VEL
LIN {X 0,Y 442.218,Z 149.445,A -85,B 0,C 180,E1 -9114.735,E2 -9114.735} C_VEL
LIN {X 0,Y 441.911,Z 145.669,A -85,B 0,C 180,E1 -9115.429,E2 -9115.429} C_VEL
LIN {X 0,Y 439.484,Z 133.745,A -85,B 0,C 180,E1 -9117.747,E2 -9117.747} C_VEL
LIN {X 0,Y 439.363,Z 133.757,A -85,B 0,C 180,E1 -9120.788,E2 -9120.788} C_VEL
LIN {X 0,Y 439.388,Z 133.756,A -85,B 0,C 180,E1 -9124.043,E2 -9124.043} C_VEL
LIN {X 0,Y 439.363,Z 133.757,A -85,B 0,C 180,E1 -9127.433,E2 -9127.433} C_VEL
LIN {X 0,Y 439.427,Z 133.752,A -85,B 0,C 180,E1 -9129.853,E2 -9129.853} C_VEL
LIN {X 0,Y 439.383,Z 133.755,A -85,B 0,C 180,E1 -9132.627,E2 -9132.627} C_VEL
LIN {X 0,Y 439.401,Z 133.751,A -85,B 0,C 180,E1 -9135.27,E2 -9135.27} C_VEL
LIN {X 0,Y 439.398,Z 133.749,A -85,B 0,C 180,E1 -9138.741,E2 -9138.741} C_VEL
LIN {X 0,Y 439.389,Z 133.751,A -85,B 0,C 180,E1 -9141.605,E2 -9141.605} C_VEL
LIN {X 0,Y 439.398,Z 133.748,A -85,B 0,C 180,E1 -9144.844,E2 -9144.844} C_VEL
LIN {X 0,Y 439.372,Z 133.755,A -85,B 0,C 180,E1 -9148.139,E2 -9148.139} C_VEL
LIN {X 0,Y 439.431,Z 133.747,A -85,B 0,C 180,E1 -9151.598,E2 -9151.598} C_VEL
LIN {X 0,Y 439.396,Z 133.746,A -85,B 0,C 180,E1 -9154.414,E2 -9154.414} C_VEL
LIN {X 0,Y 439.362,Z 133.753,A -85,B 0,C 180,E1 -9157.424,E2 -9157.424} C_VEL
LIN {X 0,Y 439.44,Z 133.74,A -85,B 0,C 180,E1 -9160.662,E2 -9160.662} C_VEL
LIN {X 0,Y 439.461,Z 133.737,A -85,B 0,C 180,E1 -9164.224,E2 -9164.224} C_VEL
LIN {X 0,Y 439.482,Z 133.736,A -85,B 0,C 180,E1 -9168.001,E2 -9168.001} C_VEL
LIN {X 0,Y 439.546,Z 133.729,A -85,B 0,C 180,E1 -9171.726,E2 -9171.726} C_VEL
LIN {X 0,Y 439.62,Z 133.722,A -85,B 0,C 180,E1 -9174.496,E2 -9174.496} C_VEL
LIN {X 0,Y 439.634,Z 133.719,A -85,B 0,C 180,E1 -9178.168,E2 -9178.168} C_VEL
LIN {X 0,Y 439.762,Z 133.701,A -85,B 0,C 180,E1 -9180,E2 -9180} C_VEL
LIN {X 0,Y 439.653,Z 133.72,A -85,B 0,C 180,E1 -9182.749,E2 -9182.749} C_VEL
LIN {X 0,Y 439.609,Z 133.722,A -85,B 0,C 180,E1 -9186.425,E2 -9186.425} C_VEL
LIN {X 0,Y 439.498,Z 133.74,A -85,B 0,C 180,E1 -9189.201,E2 -9189.201} C_VEL
LIN {X 0,Y 439.463,Z 133.746,A -85,B 0,C 180,E1 -9192.938,E2 -9192.938} C_VEL
LIN {X 0,Y 439.445,Z 133.746,A -85,B 0,C 180,E1 -9196.349,E2 -9196.349} C_VEL
LIN {X 0,Y 439.4,Z 133.749,A -85,B 0,C 180,E1 -9199.626,E2 -9199.626} C_VEL
LIN {X 0,Y 439.362,Z 133.761,A -85,B 0,C 180,E1 -9202.575,E2 -9202.575} C_VEL
LIN {X 0,Y 439.402,Z 133.753,A -85,B 0,C 180,E1 -9205.585,E2 -9205.585} C_VEL
LIN {X 0,Y 439.415,Z 133.752,A -85,B 0,C 180,E1 -9208.673,E2 -9208.673} C_VEL
LIN {X 0,Y 439.395,Z 133.755,A -85,B 0,C 180,E1 -9212.395,E2 -9212.395} C_VEL
LIN {X 0,Y 439.437,Z 133.78,A -85,B 0,C 180,E1 -9212.665,E2 -9212.665} C_VEL
LIN {X 0,Y 440.969,Z 141.603,A -85,B 0,C 180,E1 -9214.456,E2 -9214.456} C_VEL
LIN {X 0,Y 441.041,Z 143.327,A -85,B 0,C 180,E1 -9214.832,E2 -9214.832} C_VEL
LIN {X 0,Y 444.56,Z 159.057,A -85,B 0,C 180,E1 -9215.288,E2 -9215.288} C_VEL
LIN {X 0,Y 443.484,Z 250.934,A -85,B 0,C 180,E1 -9216.869,E2 -9216.869} C_VEL
LIN {X 0,Y 443.102,Z 264.652,A -85,B 0,C 180,E1 -9217.302,E2 -9217.302} C_VEL
LIN {X 0,Y 442.784,Z 276.097,A -85,B 0,C 180,E1 -9217.838,E2 -9217.838} C_VEL
LIN {X 0,Y 442.289,Z 287.707,A -85,B 0,C 180,E1 -9218.558,E2 -9218.558} C_VEL
LIN {X 0,Y 441.716,Z 299.675,A -85,B 0,C 180,E1 -9219.526,E2 -9219.526} C_VEL
LIN {X 0,Y 441.03,Z 310.427,A -85,B 0,C 180,E1 -9220.618,E2 -9220.618} C_VEL
LIN {X 0,Y 440.405,Z 319.775,A -85,B 0,C 180,E1 -9221.807,E2 -9221.807} C_VEL
LIN {X 0,Y 439.823,Z 328.045,A -85,B 0,C 180,E1 -9223.1,E2 -9223.1} C_VEL
LIN {X 0,Y 439.405,Z 334.797,A -85,B 0,C 180,E1 -9224.401,E2 -9224.401} C_VEL
LIN {X 0,Y 439.059,Z 340.257,A -85,B 0,C 180,E1 -9225.701,E2 -9225.701} C_VEL
LIN {X 0,Y 438.825,Z 344.662,A -85,B 0,C 180,E1 -9227.015,E2 -9227.015} C_VEL
LIN {X 0,Y 438.598,Z 348.058,A -85,B 0,C 180,E1 -9228.32,E2 -9228.32} C_VEL
LIN {X 0,Y 438.381,Z 351.295,A -85,B 0,C 180,E1 -9230.114,E2 -9230.114} C_VEL
LIN {X 0,Y 438.294,Z 352.851,A -85,B 0,C 180,E1 -9231.786,E2 -9231.786} C_VEL
LIN {X 0,Y 438.256,Z 353.079,A -85,B 0,C 180,E1 -9233.606,E2 -9233.606} C_VEL
LIN {X 0,Y 438.3,Z 352.308,A -85,B 0,C 180,E1 -9234.862,E2 -9234.862} C_VEL
LIN {X 0,Y 438.404,Z 350.246,A -85,B 0,C 180,E1 -9236.471,E2 -9236.471} C_VEL
LIN {X 0,Y 438.631,Z 346.787,A -85,B 0,C 180,E1 -9238.124,E2 -9238.124} C_VEL
LIN {X 0,Y 438.906,Z 341.555,A -85,B 0,C 180,E1 -9239.846,E2 -9239.846} C_VEL
LIN {X 0,Y 439.231,Z 335.675,A -85,B 0,C 180,E1 -9241.314,E2 -9241.314} C_VEL
LIN {X 0,Y 439.662,Z 329.002,A -85,B 0,C 180,E1 -9242.641,E2 -9242.641} C_VEL
LIN {X 0,Y 440.16,Z 320.815,A -85,B 0,C 180,E1 -9243.954,E2 -9243.954} C_VEL
LIN {X 0,Y 440.726,Z 311.283,A -85,B 0,C 180,E1 -9245.192,E2 -9245.192} C_VEL
LIN {X 0,Y 441.303,Z 300.839,A -85,B 0,C 180,E1 -9246.289,E2 -9246.289} C_VEL
LIN {X 0,Y 441.876,Z 290.25,A -85,B 0,C 180,E1 -9247.175,E2 -9247.175} C_VEL
LIN {X 0,Y 442.288,Z 279.827,A -85,B 0,C 180,E1 -9247.875,E2 -9247.875} C_VEL
LIN {X 0,Y 442.008,Z 274.458,A -85,B 0,C 180,E1 -9248.193,E2 -9248.193} C_VEL
LIN {X 0,Y 439.527,Z 265.692,A -85,B 0,C 180,E1 -9248.704,E2 -9248.704} C_VEL
LIN {X 0,Y 436.884,Z 256.721,A -85,B 0,C 180,E1 -9249.132,E2 -9249.132} C_VEL
LIN {X 0,Y 436.274,Z 251.028,A -85,B 0,C 180,E1 -9249.317,E2 -9249.317} C_VEL
LIN {X 0,Y 436.887,Z 200.865,A -85,B 0,C 180,E1 -9250.195,E2 -9250.195} C_VEL
LIN {X 0,Y 437.29,Z 159.685,A -85,B 0,C 180,E1 -9250.901,E2 -9250.901} C_VEL
LIN {X 0,Y 433.741,Z 142.789,A -85,B 0,C 180,E1 -9251.367,E2 -9251.367} C_VEL
LIN {X 0,Y 432.424,Z 134.622,A -85,B 0,C 180,E1 -9253.283,E2 -9253.283} C_VEL
LIN {X 0,Y 432.4,Z 134.623,A -85,B 0,C 180,E1 -9256.847,E2 -9256.847} C_VEL
LIN {X 0,Y 432.406,Z 134.625,A -85,B 0,C 180,E1 -9259.701,E2 -9259.701} C_VEL
LIN {X 0,Y 432.554,Z 134.6,A -85,B 0,C 180,E1 -9262.532,E2 -9262.532} C_VEL
LIN {X 0,Y 432.594,Z 134.595,A -85,B 0,C 180,E1 -9264.406,E2 -9264.406} C_VEL
LIN {X 0,Y 432.603,Z 134.594,A -85,B 0,C 180,E1 -9268.138,E2 -9268.138} C_VEL
LIN {X 0,Y 432.732,Z 134.579,A -85,B 0,C 180,E1 -9270,E2 -9270} C_VEL
LIN {X 0,Y 432.592,Z 134.597,A -85,B 0,C 180,E1 -9272.794,E2 -9272.794} C_VEL
LIN {X 0,Y 432.587,Z 134.599,A -85,B 0,C 180,E1 -9275.594,E2 -9275.594} C_VEL
LIN {X 0,Y 432.464,Z 134.612,A -85,B 0,C 180,E1 -9278.41,E2 -9278.41} C_VEL
LIN {X 0,Y 432.459,Z 134.612,A -85,B 0,C 180,E1 -9282.197,E2 -9282.197} C_VEL
LIN {X 0,Y 432.43,Z 134.616,A -85,B 0,C 180,E1 -9286.039,E2 -9286.039} C_VEL
LIN {X 0,Y 432.386,Z 134.622,A -85,B 0,C 180,E1 -9289.485,E2 -9289.485} C_VEL
LIN {X 0,Y 432.318,Z 134.634,A -85,B 0,C 180,E1 -9292.964,E2 -9292.964} C_VEL
LIN {X 0,Y 432.361,Z 134.625,A -85,B 0,C 180,E1 -9296.032,E2 -9296.032} C_VEL
LIN {X 0,Y 432.342,Z 134.628,A -85,B 0,C 180,E1 -9299.187,E2 -9299.187} C_VEL
LIN {X 0,Y 432.321,Z 134.635,A -85,B 0,C 180,E1 -9302.443,E2 -9302.443} C_VEL
LIN {X 0,Y 432.341,Z 134.627,A -85,B 0,C 180,E1 -9305.631,E2 -9305.631} C_VEL
LIN {X 0,Y 432.336,Z 134.631,A -85,B 0,C 180,E1 -9308.714,E2 -9308.714} C_VEL
LIN {X 0,Y 432.332,Z 134.63,A -85,B 0,C 180,E1 -9311.797,E2 -9311.797} C_VEL
LIN {X 0,Y 432.332,Z 134.634,A -85,B 0,C 180,E1 -9314.347,E2 -9314.347} C_VEL
LIN {X 0,Y 432.318,Z 134.63,A -85,B 0,C 180,E1 -9317.016,E2 -9317.016} C_VEL
LIN {X 0,Y 432.339,Z 134.631,A -85,B 0,C 180,E1 -9319.819,E2 -9319.819} C_VEL
LIN {X 0,Y 432.313,Z 134.63,A -85,B 0,C 180,E1 -9323.023,E2 -9323.023} C_VEL
LIN {X 0,Y 432.358,Z 134.632,A -85,B 0,C 180,E1 -9325.996,E2 -9325.996} C_VEL
LIN {X 0,Y 432.346,Z 134.629,A -85,B 0,C 180,E1 -9329.49,E2 -9329.49} C_VEL
LIN {X 0,Y 432.388,Z 134.621,A -85,B 0,C 180,E1 -9332.928,E2 -9332.928} C_VEL
LIN {X 0,Y 432.366,Z 134.627,A -85,B 0,C 180,E1 -9336.023,E2 -9336.023} C_VEL
LIN {X 0,Y 432.348,Z 134.627,A -85,B 0,C 180,E1 -9339.046,E2 -9339.046} C_VEL
LIN {X 0,Y 432.376,Z 134.624,A -85,B 0,C 180,E1 -9342.011,E2 -9342.011} C_VEL
LIN {X 0,Y 432.395,Z 134.621,A -85,B 0,C 180,E1 -9344.927,E2 -9344.927} C_VEL
LIN {X 0,Y 432.457,Z 134.615,A -85,B 0,C 180,E1 -9347.804,E2 -9347.804} C_VEL
LIN {X 0,Y 432.49,Z 134.612,A -85,B 0,C 180,E1 -9351.59,E2 -9351.59} C_VEL
LIN {X 0,Y 432.597,Z 134.595,A -85,B 0,C 180,E1 -9354.406,E2 -9354.406} C_VEL
LIN {X 0,Y 432.604,Z 134.594,A -85,B 0,C 180,E1 -9358.138,E2 -9358.138} C_VEL
LIN {X 0,Y 432.732,Z 134.578,A -85,B 0,C 180,E1 -9360,E2 -9360} C_VEL
LIN {X 0,Y 432.603,Z 134.598,A -85,B 0,C 180,E1 -9362.794,E2 -9362.794} C_VEL
LIN {X 0,Y 432.563,Z 134.602,A -85,B 0,C 180,E1 -9366.531,E2 -9366.531} C_VEL
LIN {X 0,Y 432.442,Z 134.616,A -85,B 0,C 180,E1 -9369.353,E2 -9369.353} C_VEL
LIN {X 0,Y 432.43,Z 134.623,A -85,B 0,C 180,E1 -9372.804,E2 -9372.804} C_VEL
LIN {X 0,Y 432.412,Z 134.623,A -85,B 0,C 180,E1 -9376.479,E2 -9376.479} C_VEL
LIN {X 0,Y 432.338,Z 134.628,A -85,B 0,C 180,E1 -9379.961,E2 -9379.961} C_VEL
LIN {X 0,Y 432.318,Z 134.632,A -85,B 0,C 180,E1 -9382.965,E2 -9382.965} C_VEL
LIN {X 0,Y 432.363,Z 134.626,A -85,B 0,C 180,E1 -9386.033,E2 -9386.033} C_VEL
LIN {X 0,Y 432.342,Z 134.627,A -85,B 0,C 180,E1 -9389.188,E2 -9389.188} C_VEL
LIN {X 0,Y 432.322,Z 134.634,A -85,B 0,C 180,E1 -9392.443,E2 -9392.443} C_VEL
LIN {X 0,Y 432.344,Z 134.627,A -85,B 0,C 180,E1 -9395.632,E2 -9395.632} C_VEL
LIN {X 0,Y 432.358,Z 134.626,A -85,B 0,C 180,E1 -9398.718,E2 -9398.718} C_VEL
LIN {X 0,Y 432.366,Z 134.628,A -85,B 0,C 180,E1 -9401.794,E2 -9401.794} C_VEL
LIN {X 0,Y 432.334,Z 134.631,A -85,B 0,C 180,E1 -9404.348,E2 -9404.348} C_VEL
LIN {X 0,Y 432.321,Z 134.629,A -85,B 0,C 180,E1 -9407.016,E2 -9407.016} C_VEL
LIN {X 0,Y 432.357,Z 134.632,A -85,B 0,C 180,E1 -9409.818,E2 -9409.818} C_VEL
LIN {X 0,Y 432.317,Z 134.63,A -85,B 0,C 180,E1 -9413.023,E2 -9413.023} C_VEL
LIN {X 0,Y 432.361,Z 134.631,A -85,B 0,C 180,E1 -9415.997,E2 -9415.997} C_VEL
LIN {X 0,Y 432.349,Z 134.632,A -85,B 0,C 180,E1 -9419.49,E2 -9419.49} C_VEL
LIN {X 0,Y 432.442,Z 134.749,A -85,B 0,C 180,E1 -9421.98,E2 -9421.98} C_VEL
LIN {X 0,Y 435.245,Z 148.696,A -85,B 0,C 180,E1 -9424.722,E2 -9424.722} C_VEL
LIN {X 0,Y 435.062,Z 155.34,A -85,B 0,C 180,E1 -9425.928,E2 -9425.928} C_VEL
LIN {X 0,Y 434.247,Z 169.188,A -85,B 0,C 180,E1 -9428.396,E2 -9428.396} C_VEL
LIN {X 0,Y 433.535,Z 184.38,A -85,B 0,C 180,E1 -9431.082,E2 -9431.082} C_VEL
LIN {X 0,Y 433.352,Z 187.569,A -85,B 0,C 180,E1 -9431.641,E2 -9431.641} C_VEL
LIN {X 0,Y 436.966,Z 214.012,A -85,B 0,C 180,E1 -9432.262,E2 -9432.262} C_VEL
LIN {X 0,Y 436.072,Z 296.279,A -85,B 0,C 180,E1 -9433.678,E2 -9433.678} C_VEL
LIN {X 0,Y 435.576,Z 309.494,A -85,B 0,C 180,E1 -9434.08,E2 -9434.08} C_VEL
LIN {X 0,Y 434.997,Z 322.238,A -85,B 0,C 180,E1 -9434.659,E2 -9434.659} C_VEL
LIN {X 0,Y 434.373,Z 333.596,A -85,B 0,C 180,E1 -9435.356,E2 -9435.356} C_VEL
LIN {X 0,Y 433.742,Z 345.083,A -85,B 0,C 180,E1 -9436.27,E2 -9436.27} C_VEL
LIN {X 0,Y 433.058,Z 355.879,A -85,B 0,C 180,E1 -9437.345,E2 -9437.345} C_VEL
LIN {X 0,Y 432.522,Z 365.393,A -85,B 0,C 180,E1 -9438.519,E2 -9438.519} C_VEL
LIN {X 0,Y 431.932,Z 374.552,A -85,B 0,C 180,E1 -9439.926,E2 -9439.926} C_VEL
LIN {X 0,Y 431.63,Z 381.941,A -85,B 0,C 180,E1 -9441.338,E2 -9441.338} C_VEL
LIN {X 0,Y 431.426,Z 386.94,A -85,B 0,C 180,E1 -9442.512,E2 -9442.512} C_VEL
LIN {X 0,Y 431.256,Z 392.211,A -85,B 0,C 180,E1 -9444.057,E2 -9444.057} C_VEL
LIN {X 0,Y 431.279,Z 395.501,A -85,B 0,C 180,E1 -9445.326,E2 -9445.326} C_VEL
LIN {X 0,Y 431.241,Z 397.412,A -85,B 0,C 180,E1 -9446.262,E2 -9446.262} C_VEL
LIN {X 0,Y 431.327,Z 398.868,A -85,B 0,C 180,E1 -9447.198,E2 -9447.198} C_VEL
LIN {X 0,Y 431.285,Z 400.507,A -85,B 0,C 180,E1 -9449.066,E2 -9449.066} C_VEL
LIN {X 0,Y 431.294,Z 400.737,A -85,B 0,C 180,E1 -9450,E2 -9450} C_VEL
LIN {X 0,Y 431.269,Z 400.531,A -85,B 0,C 180,E1 -9450.934,E2 -9450.934} C_VEL
LIN {X 0,Y 431.326,Z 398.901,A -85,B 0,C 180,E1 -9452.802,E2 -9452.802} C_VEL
LIN {X 0,Y 431.238,Z 397.48,A -85,B 0,C 180,E1 -9453.738,E2 -9453.738} C_VEL
LIN {X 0,Y 431.31,Z 394.5,A -85,B 0,C 180,E1 -9455.142,E2 -9455.142} C_VEL
LIN {X 0,Y 431.291,Z 390.466,A -85,B 0,C 180,E1 -9456.55,E2 -9456.55} C_VEL
LIN {X 0,Y 431.565,Z 384.289,A -85,B 0,C 180,E1 -9458.192,E2 -9458.192} C_VEL
LIN {X 0,Y 431.829,Z 377.531,A -85,B 0,C 180,E1 -9459.603,E2 -9459.603} C_VEL
LIN {X 0,Y 432.322,Z 369.163,A -85,B 0,C 180,E1 -9461.012,E2 -9461.012} C_VEL
LIN {X 0,Y 432.873,Z 360.615,A -85,B 0,C 180,E1 -9462.185,E2 -9462.185} C_VEL
LIN {X 0,Y 433.504,Z 350.341,A -85,B 0,C 180,E1 -9463.33,E2 -9463.33} C_VEL
LIN {X 0,Y 434.135,Z 339.665,A -85,B 0,C 180,E1 -9464.293,E2 -9464.293} C_VEL
LIN {X 0,Y 434.877,Z 328.295,A -85,B 0,C 180,E1 -9465.105,E2 -9465.105} C_VEL
LIN {X 0,Y 435.509,Z 316.719,A -85,B 0,C 180,E1 -9465.742,E2 -9465.742} C_VEL
LIN {X 0,Y 436.066,Z 304.398,A -85,B 0,C 180,E1 -9466.232,E2 -9466.232} C_VEL
LIN {X 0,Y 436.519,Z 290.81,A -85,B 0,C 180,E1 -9466.575,E2 -9466.575} C_VEL
LIN {X 0,Y 437.2,Z 212.537,A -85,B 0,C 180,E1 -9467.928,E2 -9467.928} C_VEL
LIN {X 0,Y 433.993,Z 190.104,A -85,B 0,C 180,E1 -9468.474,E2 -9468.474} C_VEL
LIN {X 0,Y 433.406,Z 186.336,A -85,B 0,C 180,E1 -9468.587,E2 -9468.587} C_VEL
LIN {X 0,Y 434.329,Z 167.727,A -85,B 0,C 180,E1 -9471.849,E2 -9471.849} C_VEL
LIN {X 0,Y 435.302,Z 150.991,A -85,B 0,C 180,E1 -9474.82,E2 -9474.82} C_VEL
LIN {X 0,Y 434.877,Z 146.363,A -85,B 0,C 180,E1 -9475.688,E2 -9475.688} C_VEL
LIN {X 0,Y 432.428,Z 134.624,A -85,B 0,C 180,E1 -9478.054,E2 -9478.054} C_VEL
LIN {X 0,Y 432.322,Z 134.632,A -85,B 0,C 180,E1 -9481.346,E2 -9481.346} C_VEL
LIN {X 0,Y 432.341,Z 134.633,A -85,B 0,C 180,E1 -9484.677,E2 -9484.677} C_VEL
LIN {X 0,Y 432.351,Z 134.637,A -85,B 0,C 180,E1 -9488.148,E2 -9488.148} C_VEL
LIN {X 0,Y 432.367,Z 134.628,A -85,B 0,C 180,E1 -9491.607,E2 -9491.607} C_VEL
LIN {X 0,Y 432.334,Z 134.636,A -85,B 0,C 180,E1 -9494.347,E2 -9494.347} C_VEL
LIN {X 0,Y 432.32,Z 134.633,A -85,B 0,C 180,E1 -9497.015,E2 -9497.015} C_VEL
LIN {X 0,Y 432.355,Z 134.632,A -85,B 0,C 180,E1 -9499.817,E2 -9499.817} C_VEL
LIN {X 0,Y 432.315,Z 134.632,A -85,B 0,C 180,E1 -9503.023,E2 -9503.023} C_VEL
LIN {X 0,Y 432.358,Z 134.629,A -85,B 0,C 180,E1 -9505.996,E2 -9505.996} C_VEL
LIN {X 0,Y 432.346,Z 134.632,A -85,B 0,C 180,E1 -9509.489,E2 -9509.489} C_VEL
LIN {X 0,Y 432.389,Z 134.621,A -85,B 0,C 180,E1 -9512.928,E2 -9512.928} C_VEL
LIN {X 0,Y 432.366,Z 134.624,A -85,B 0,C 180,E1 -9516.023,E2 -9516.023} C_VEL
LIN {X 0,Y 432.349,Z 134.626,A -85,B 0,C 180,E1 -9519.046,E2 -9519.046} C_VEL
LIN {X 0,Y 432.377,Z 134.623,A -85,B 0,C 180,E1 -9522.011,E2 -9522.011} C_VEL
LIN {X 0,Y 432.395,Z 134.619,A -85,B 0,C 180,E1 -9524.926,E2 -9524.926} C_VEL
LIN {X 0,Y 432.458,Z 134.612,A -85,B 0,C 180,E1 -9527.803,E2 -9527.803} C_VEL
LIN {X 0,Y 432.49,Z 134.609,A -85,B 0,C 180,E1 -9531.59,E2 -9531.59} C_VEL
LIN {X 0,Y 432.597,Z 134.596,A -85,B 0,C 180,E1 -9534.406,E2 -9534.406} C_VEL
LIN {X 0,Y 432.604,Z 134.595,A -85,B 0,C 180,E1 -9538.138,E2 -9538.138} C_VEL
LIN {X 0,Y 432.732,Z 134.576,A -85,B 0,C 180,E1 -9540,E2 -9540} C_VEL
LIN {X 0,Y 432.603,Z 134.598,A -85,B 0,C 180,E1 -9542.793,E2 -9542.793} C_VEL
LIN {X 0,Y 432.562,Z 134.6,A -85,B 0,C 180,E1 -9546.53,E2 -9546.53} C_VEL
LIN {X 0,Y 432.441,Z 134.618,A -85,B 0,C 180,E1 -9549.353,E2 -9549.353} C_VEL
LIN {X 0,Y 432.428,Z 134.624,A -85,B 0,C 180,E1 -9552.803,E2 -9552.803} C_VEL
LIN {X 0,Y 432.41,Z 134.623,A -85,B 0,C 180,E1 -9556.479,E2 -9556.479} C_VEL
LIN {X 0,Y 432.337,Z 134.63,A -85,B 0,C 180,E1 -9559.96,E2 -9559.96} C_VEL
LIN {X 0,Y 432.316,Z 134.638,A -85,B 0,C 180,E1 -9562.964,E2 -9562.964} C_VEL
LIN {X 0,Y 432.362,Z 134.631,A -85,B 0,C 180,E1 -9566.032,E2 -9566.032} C_VEL
LIN {X 0,Y 432.341,Z 134.631,A -85,B 0,C 180,E1 -9569.187,E2 -9569.187} C_VEL
LIN {X 0,Y 432.391,Z 134.799,A -85,B 0,C 180,E1 -9572.437,E2 -9572.437} C_VEL
LIN {X 0,Y 434.125,Z 143.746,A -85,B 0,C 180,E1 -9574.514,E2 -9574.514} C_VEL
LIN {X 0,Y 437.793,Z 159.769,A -85,B 0,C 180,E1 -9574.992,E2 -9574.992} C_VEL
LIN {X 0,Y 436.72,Z 251.336,A -85,B 0,C 180,E1 -9576.597,E2 -9576.597} C_VEL
LIN {X 0,Y 436.343,Z 264.854,A -85,B 0,C 180,E1 -9577.03,E2 -9577.03} C_VEL
LIN {X 0,Y 435.981,Z 276.618,A -85,B 0,C 180,E1 -9577.587,E2 -9577.587} C_VEL
LIN {X 0,Y 435.442,Z 288.521,A -85,B 0,C 180,E1 -9578.343,E2 -9578.343} C_VEL
LIN {X 0,Y 434.919,Z 299.041,A -85,B 0,C 180,E1 -9579.2,E2 -9579.2} C_VEL
LIN {X 0,Y 434.22,Z 308.989,A -85,B 0,C 180,E1 -9580.197,E2 -9580.197} C_VEL
LIN {X 0,Y 433.57,Z 318.894,A -85,B 0,C 180,E1 -9581.427,E2 -9581.427} C_VEL
LIN {X 0,Y 432.941,Z 327.333,A -85,B 0,C 180,E1 -9582.732,E2 -9582.732} C_VEL
LIN {X 0,Y 432.474,Z 334.124,A -85,B 0,C 180,E1 -9584.021,E2 -9584.021} C_VEL
LIN {X 0,Y 432.034,Z 340.826,A -85,B 0,C 180,E1 -9585.614,E2 -9585.614} C_VEL
LIN {X 0,Y 431.748,Z 345.632,A -85,B 0,C 180,E1 -9587.097,E2 -9587.097} C_VEL
LIN {X 0,Y 431.511,Z 349.1,A -85,B 0,C 180,E1 -9588.521,E2 -9588.521} C_VEL
LIN {X 0,Y 431.327,Z 351.591,A -85,B 0,C 180,E1 -9589.979,E2 -9589.979} C_VEL
LIN {X 0,Y 431.21,Z 353.233,A -85,B 0,C 180,E1 -9591.733,E2 -9591.733} C_VEL
LIN {X 0,Y 431.197,Z 353.58,A -85,B 0,C 180,E1 -9593,E2 -9593} C_VEL
LIN {X 0,Y 431.191,Z 352.955,A -85,B 0,C 180,E1 -9594.582,E2 -9594.582} C_VEL
LIN {X 0,Y 431.307,Z 350.874,A -85,B 0,C 180,E1 -9596.357,E2 -9596.357} C_VEL
LIN {X 0,Y 431.529,Z 347.913,A -85,B 0,C 180,E1 -9597.874,E2 -9597.874} C_VEL
LIN {X 0,Y 431.776,Z 343.051,A -85,B 0,C 180,E1 -9599.618,E2 -9599.618} C_VEL
LIN {X 0,Y 432.166,Z 337.273,A -85,B 0,C 180,E1 -9601.148,E2 -9601.148} C_VEL
LIN {X 0,Y 432.613,Z 329.9,A -85,B 0,C 180,E1 -9602.682,E2 -9602.682} C_VEL
LIN {X 0,Y 433.146,Z 321.854,A -85,B 0,C 180,E1 -9604.018,E2 -9604.018} C_VEL
LIN {X 0,Y 433.662,Z 313.357,A -85,B 0,C 180,E1 -9605.168,E2 -9605.168} C_VEL
LIN {X 0,Y 434.248,Z 303.481,A -85,B 0,C 180,E1 -9606.261,E2 -9606.261} C_VEL
LIN {X 0,Y 434.82,Z 293.289,A -85,B 0,C 180,E1 -9607.176,E2 -9607.176} C_VEL
LIN {X 0,Y 435.353,Z 281.512,A -85,B 0,C 180,E1 -9608.018,E2 -9608.018} C_VEL
LIN {X 0,Y 435.799,Z 269.538,A -85,B 0,C 180,E1 -9608.663,E2 -9608.663} C_VEL
LIN {X 0,Y 436.2,Z 256.652,A -85,B 0,C 180,E1 -9609.158,E2 -9609.158} C_VEL
LIN {X 0,Y 436.274,Z 251.028,A -85,B 0,C 180,E1 -9609.317,E2 -9609.317} C_VEL
LIN {X 0,Y 435.719,Z 245.263,A -85,B 0,C 180,E1 -9609.475,E2 -9609.475} C_VEL
LIN {X 0,Y 430.374,Z 226.555,A -85,B 0,C 180,E1 -9609.998,E2 -9609.998} C_VEL
LIN {X 0,Y 429.816,Z 220.738,A -85,B 0,C 180,E1 -9610.117,E2 -9610.117} C_VEL
LIN {X 0,Y 430.527,Z 160.813,A -85,B 0,C 180,E1 -9611.158,E2 -9611.158} C_VEL
LIN {X 0,Y 426.705,Z 143.167,A -85,B 0,C 180,E1 -9611.657,E2 -9611.657} C_VEL
LIN {X 0,Y 425.395,Z 135.499,A -85,B 0,C 180,E1 -9613.518,E2 -9613.518} C_VEL
LIN {X 0,Y 425.393,Z 135.497,A -85,B 0,C 180,E1 -9617.096,E2 -9617.096} C_VEL
LIN {X 0,Y 425.4,Z 135.491,A -85,B 0,C 180,E1 -9620.491,E2 -9620.491} C_VEL
LIN {X 0,Y 425.523,Z 135.481,A -85,B 0,C 180,E1 -9623.361,E2 -9623.361} C_VEL
LIN {X 0,Y 425.366,Z 135.5,A -85,B 0,C 180,E1 -9625.261,E2 -9625.261} C_VEL
LIN {X 0,Y 425.572,Z 135.47,A -85,B 0,C 180,E1 -9628.107,E2 -9628.107} C_VEL
LIN {X 0,Y 425.702,Z 135.455,A -85,B 0,C 180,E1 -9630,E2 -9630} C_VEL
LIN {X 0,Y 425.545,Z 135.476,A -85,B 0,C 180,E1 -9632.84,E2 -9632.84} C_VEL
LIN {X 0,Y 425.542,Z 135.476,A -85,B 0,C 180,E1 -9635.687,E2 -9635.687} C_VEL
LIN {X 0,Y 425.408,Z 135.492,A -85,B 0,C 180,E1 -9638.551,E2 -9638.551} C_VEL
LIN {X 0,Y 425.412,Z 135.491,A -85,B 0,C 180,E1 -9642.402,E2 -9642.402} C_VEL
LIN {X 0,Y 425.388,Z 135.494,A -85,B 0,C 180,E1 -9646.312,E2 -9646.312} C_VEL
LIN {X 0,Y 425.328,Z 135.501,A -85,B 0,C 180,E1 -9649.635,E2 -9649.635} C_VEL
LIN {X 0,Y 425.287,Z 135.508,A -85,B 0,C 180,E1 -9652.339,E2 -9652.339} C_VEL
LIN {X 0,Y 425.292,Z 135.505,A -85,B 0,C 180,E1 -9655.445,E2 -9655.445} C_VEL
LIN {X 0,Y 425.33,Z 135.508,A -85,B 0,C 180,E1 -9658.632,E2 -9658.632} C_VEL
LIN {X 0,Y 425.263,Z 135.509,A -85,B 0,C 180,E1 -9661.927,E2 -9661.927} C_VEL
LIN {X 0,Y 425.296,Z 135.504,A -85,B 0,C 180,E1 -9665.336,E2 -9665.336} C_VEL
LIN {X 0,Y 425.295,Z 135.506,A -85,B 0,C 180,E1 -9668.899,E2 -9668.899} C_VEL
LIN {X 0,Y 425.288,Z 135.508,A -85,B 0,C 180,E1 -9671.958,E2 -9671.958} C_VEL
LIN {X 0,Y 425.285,Z 135.506,A -85,B 0,C 180,E1 -9675.283,E2 -9675.283} C_VEL
LIN {X 0,Y 425.273,Z 135.509,A -85,B 0,C 180,E1 -9678.621,E2 -9678.621} C_VEL
LIN {X 0,Y 425.314,Z 135.502,A -85,B 0,C 180,E1 -9681.103,E2 -9681.103} C_VEL
LIN {X 0,Y 425.298,Z 135.505,A -85,B 0,C 180,E1 -9684.664,E2 -9684.664} C_VEL
LIN {X 0,Y 425.264,Z 135.513,A -85,B 0,C 180,E1 -9688.073,E2 -9688.073} C_VEL
LIN {X 0,Y 425.329,Z 135.502,A -85,B 0,C 180,E1 -9691.368,E2 -9691.368} C_VEL
LIN {X 0,Y 425.351,Z 135.501,A -85,B 0,C 180,E1 -9693.505,E2 -9693.505} C_VEL
LIN {X 0,Y 425.283,Z 135.506,A -85,B 0,C 180,E1 -9696.634,E2 -9696.634} C_VEL
LIN {X 0,Y 425.293,Z 135.511,A -85,B 0,C 180,E1 -9699.695,E2 -9699.695} C_VEL
LIN {X 0,Y 425.34,Z 135.499,A -85,B 0,C 180,E1 -9702.698,E2 -9702.698} C_VEL
LIN {X 0,Y 425.347,Z 135.503,A -85,B 0,C 180,E1 -9705.65,E2 -9705.65} C_VEL
LIN {X 0,Y 425.35,Z 135.498,A -85,B 0,C 180,E1 -9708.564,E2 -9708.564} C_VEL
LIN {X 0,Y 425.536,Z 135.474,A -85,B 0,C 180,E1 -9712.408,E2 -9712.408} C_VEL
LIN {X 0,Y 425.554,Z 135.472,A -85,B 0,C 180,E1 -9714.313,E2 -9714.313} C_VEL
LIN {X 0,Y 425.573,Z 135.47,A -85,B 0,C 180,E1 -9718.107,E2 -9718.107} C_VEL
LIN {X 0,Y 425.702,Z 135.454,A -85,B 0,C 180,E1 -9720,E2 -9720} C_VEL
LIN {X 0,Y 425.555,Z 135.477,A -85,B 0,C 180,E1 -9722.84,E2 -9722.84} C_VEL
LIN {X 0,Y 425.522,Z 135.48,A -85,B 0,C 180,E1 -9726.639,E2 -9726.639} C_VEL
LIN {X 0,Y 425.4,Z 135.492,A -85,B 0,C 180,E1 -9729.51,E2 -9729.51} C_VEL
LIN {X 0,Y 425.392,Z 135.498,A -85,B 0,C 180,E1 -9732.904,E2 -9732.904} C_VEL
LIN {X 0,Y 425.361,Z 135.503,A -85,B 0,C 180,E1 -9736.605,E2 -9736.605} C_VEL
LIN {X 0,Y 425.328,Z 135.5,A -85,B 0,C 180,E1 -9739.636,E2 -9739.636} C_VEL
LIN {X 0,Y 425.287,Z 135.51,A -85,B 0,C 180,E1 -9742.339,E2 -9742.339} C_VEL
LIN {X 0,Y 425.294,Z 135.504,A -85,B 0,C 180,E1 -9745.446,E2 -9745.446} C_VEL
LIN {X 0,Y 425.331,Z 135.504,A -85,B 0,C 180,E1 -9748.632,E2 -9748.632} C_VEL
LIN {X 0,Y 425.264,Z 135.511,A -85,B 0,C 180,E1 -9751.927,E2 -9751.927} C_VEL
LIN {X 0,Y 425.299,Z 135.504,A -85,B 0,C 180,E1 -9755.336,E2 -9755.336} C_VEL
LIN {X 0,Y 425.311,Z 135.502,A -85,B 0,C 180,E1 -9759.046,E2 -9759.046} C_VEL
LIN {X 0,Y 425.316,Z 135.508,A -85,B 0,C 180,E1 -9761.962,E2 -9761.962} C_VEL
LIN {X 0,Y 425.285,Z 135.506,A -85,B 0,C 180,E1 -9765.283,E2 -9765.283} C_VEL
LIN {X 0,Y 425.305,Z 135.504,A -85,B 0,C 180,E1 -9768.625,E2 -9768.625} C_VEL
LIN {X 0,Y 425.323,Z 135.501,A -85,B 0,C 180,E1 -9771.104,E2 -9771.104} C_VEL
LIN {X 0,Y 425.301,Z 135.504,A -85,B 0,C 180,E1 -9774.664,E2 -9774.664} C_VEL
LIN {X 0,Y 425.266,Z 135.511,A -85,B 0,C 180,E1 -9778.073,E2 -9778.073} C_VEL
LIN {X 0,Y 425.379,Z 135.634,A -85,B 0,C 180,E1 -9781.742,E2 -9781.742} C_VEL
LIN {X 0,Y 428.199,Z 149.492,A -85,B 0,C 180,E1 -9784.517,E2 -9784.517} C_VEL
LIN {X 0,Y 428.355,Z 153.48,A -85,B 0,C 180,E1 -9785.268,E2 -9785.268} C_VEL
LIN {X 0,Y 427.274,Z 170.098,A -85,B 0,C 180,E1 -9788.279,E2 -9788.279} C_VEL
LIN {X 0,Y 426.606,Z 183.915,A -85,B 0,C 180,E1 -9790.763,E2 -9790.763} C_VEL
LIN {X 0,Y 426.381,Z 187.253,A -85,B 0,C 180,E1 -9791.357,E2 -9791.357} C_VEL
LIN {X 0,Y 430.155,Z 214.664,A -85,B 0,C 180,E1 -9792.007,E2 -9792.007} C_VEL
LIN {X 0,Y 429.202,Z 296.247,A -85,B 0,C 180,E1 -9793.44,E2 -9793.44} C_VEL
LIN {X 0,Y 428.705,Z 309.347,A -85,B 0,C 180,E1 -9793.849,E2 -9793.849} C_VEL
LIN {X 0,Y 428.139,Z 321.47,A -85,B 0,C 180,E1 -9794.407,E2 -9794.407} C_VEL
LIN {X 0,Y 427.491,Z 332.936,A -85,B 0,C 180,E1 -9795.115,E2 -9795.115} C_VEL
LIN {X 0,Y 426.785,Z 344.737,A -85,B 0,C 180,E1 -9796.065,E2 -9796.065} C_VEL
LIN {X 0,Y 426.101,Z 355.325,A -85,B 0,C 180,E1 -9797.134,E2 -9797.134} C_VEL
LIN {X 0,Y 425.527,Z 364.877,A -85,B 0,C 180,E1 -9798.327,E2 -9798.327} C_VEL
LIN {X 0,Y 424.877,Z 374.061,A -85,B 0,C 180,E1 -9799.757,E2 -9799.757} C_VEL
LIN {X 0,Y 424.542,Z 381.47,A -85,B 0,C 180,E1 -9801.192,E2 -9801.192} C_VEL
LIN {X 0,Y 424.353,Z 386.487,A -85,B 0,C 180,E1 -9802.386,E2 -9802.386} C_VEL
LIN {X 0,Y 424.227,Z 391.056,A -85,B 0,C 180,E1 -9803.72,E2 -9803.72} C_VEL
LIN {X 0,Y 424.209,Z 395.079,A -85,B 0,C 180,E1 -9805.248,E2 -9805.248} C_VEL
LIN {X 0,Y 424.147,Z 396.995,A -85,B 0,C 180,E1 -9806.2,E2 -9806.2} C_VEL
LIN {X 0,Y 424.253,Z 398.464,A -85,B 0,C 180,E1 -9807.151,E2 -9807.151} C_VEL
LIN {X 0,Y 424.198,Z 400.112,A -85,B 0,C 180,E1 -9809.051,E2 -9809.051} C_VEL
LIN {X 0,Y 424.204,Z 400.345,A -85,B 0,C 180,E1 -9810,E2 -9810} C_VEL
LIN {X 0,Y 424.183,Z 400.148,A -85,B 0,C 180,E1 -9810.949,E2 -9810.949} C_VEL
LIN {X 0,Y 424.235,Z 398.524,A -85,B 0,C 180,E1 -9812.849,E2 -9812.849} C_VEL
LIN {X 0,Y 424.145,Z 397.105,A -85,B 0,C 180,E1 -9813.8,E2 -9813.8} C_VEL
LIN {X 0,Y 424.217,Z 394.131,A -85,B 0,C 180,E1 -9815.228,E2 -9815.228} C_VEL
LIN {X 0,Y 424.225,Z 390.104,A -85,B 0,C 180,E1 -9816.659,E2 -9816.659} C_VEL
LIN {X 0,Y 424.494,Z 383.942,A -85,B 0,C 180,E1 -9818.329,E2 -9818.329} C_VEL
LIN {X 0,Y 424.8,Z 377.2,A -85,B 0,C 180,E1 -9819.763,E2 -9819.763} C_VEL
LIN {X 0,Y 425.325,Z 368.851,A -85,B 0,C 180,E1 -9821.195,E2 -9821.195} C_VEL
LIN {X 0,Y 425.88,Z 360.321,A -85,B 0,C 180,E1 -9822.388,E2 -9822.388} C_VEL
LIN {X 0,Y 426.572,Z 349.831,A -85,B 0,C 180,E1 -9823.576,E2 -9823.576} C_VEL
LIN {X 0,Y 427.346,Z 337.993,A -85,B 0,C 180,E1 -9824.646,E2 -9824.646} C_VEL
LIN {X 0,Y 428.11,Z 326.218,A -85,B 0,C 180,E1 -9825.472,E2 -9825.472} C_VEL
LIN {X 0,Y 428.856,Z 312.733,A -85,B 0,C 180,E1 -9826.176,E2 -9826.176} C_VEL
LIN {X 0,Y 429.449,Z 299.815,A -85,B 0,C 180,E1 -9826.642,E2 -9826.642} C_VEL
LIN {X 0,Y 429.776,Z 286.269,A -85,B 0,C 180,E1 -9826.935,E2 -9826.935} C_VEL
LIN {X 0,Y 430.446,Z 213.16,A -85,B 0,C 180,E1 -9828.22,E2 -9828.22} C_VEL
LIN {X 0,Y 427.234,Z 190.495,A -85,B 0,C 180,E1 -9828.787,E2 -9828.787} C_VEL
LIN {X 0,Y 426.496,Z 185.854,A -85,B 0,C 180,E1 -9828.933,E2 -9828.933} C_VEL
LIN {X 0,Y 427.577,Z 166.265,A -85,B 0,C 180,E1 -9832.429,E2 -9832.429} C_VEL
LIN {X 0,Y 428.432,Z 150.705,A -85,B 0,C 180,E1 -9835.246,E2 -9835.246} C_VEL
LIN {X 0,Y 426.259,Z 139.452,A -85,B 0,C 180,E1 -9837.494,E2 -9837.494} C_VEL
LIN {X 0,Y 425.35,Z 135.506,A -85,B 0,C 180,E1 -9838.328,E2 -9838.328} C_VEL
LIN {X 0,Y 425.266,Z 135.514,A -85,B 0,C 180,E1 -9841.927,E2 -9841.927} C_VEL
LIN {X 0,Y 425.3,Z 135.507,A -85,B 0,C 180,E1 -9845.335,E2 -9845.335} C_VEL
LIN {X 0,Y 425.311,Z 135.508,A -85,B 0,C 180,E1 -9849.045,E2 -9849.045} C_VEL
LIN {X 0,Y 425.316,Z 135.511,A -85,B 0,C 180,E1 -9851.962,E2 -9851.962} C_VEL
LIN {X 0,Y 425.285,Z 135.51,A -85,B 0,C 180,E1 -9855.283,E2 -9855.283} C_VEL
LIN {X 0,Y 425.304,Z 135.506,A -85,B 0,C 180,E1 -9858.625,E2 -9858.625} C_VEL
LIN {X 0,Y 425.321,Z 135.501,A -85,B 0,C 180,E1 -9861.104,E2 -9861.104} C_VEL
LIN {X 0,Y 425.299,Z 135.505,A -85,B 0,C 180,E1 -9864.664,E2 -9864.664} C_VEL
LIN {X 0,Y 425.264,Z 135.513,A -85,B 0,C 180,E1 -9868.073,E2 -9868.073} C_VEL
LIN {X 0,Y 425.33,Z 135.501,A -85,B 0,C 180,E1 -9871.368,E2 -9871.368} C_VEL
LIN {X 0,Y 425.352,Z 135.499,A -85,B 0,C 180,E1 -9873.505,E2 -9873.505} C_VEL
LIN {X 0,Y 425.283,Z 135.504,A -85,B 0,C 180,E1 -9876.633,E2 -9876.633} C_VEL
LIN {X 0,Y 425.294,Z 135.507,A -85,B 0,C 180,E1 -9879.694,E2 -9879.694} C_VEL
LIN {X 0,Y 425.341,Z 135.498,A -85,B 0,C 180,E1 -9882.697,E2 -9882.697} C_VEL
LIN {X 0,Y 425.348,Z 135.502,A -85,B 0,C 180,E1 -9885.65,E2 -9885.65} C_VEL
LIN {X 0,Y 425.35,Z 135.496,A -85,B 0,C 180,E1 -9888.564,E2 -9888.564} C_VEL
LIN {X 0,Y 425.536,Z 135.472,A -85,B 0,C 180,E1 -9892.407,E2 -9892.407} C_VEL
LIN {X 0,Y 425.553,Z 135.474,A -85,B 0,C 180,E1 -9894.313,E2 -9894.313} C_VEL
LIN {X 0,Y 425.573,Z 135.471,A -85,B 0,C 180,E1 -9898.107,E2 -9898.107} C_VEL
LIN {X 0,Y 425.701,Z 135.452,A -85,B 0,C 180,E1 -9900,E2 -9900} C_VEL
LIN {X 0,Y 425.554,Z 135.475,A -85,B 0,C 180,E1 -9902.84,E2 -9902.84} C_VEL
LIN {X 0,Y 425.521,Z 135.478,A -85,B 0,C 180,E1 -9906.639,E2 -9906.639} C_VEL
LIN {X 0,Y 425.399,Z 135.494,A -85,B 0,C 180,E1 -9909.509,E2 -9909.509} C_VEL
LIN {X 0,Y 425.391,Z 135.499,A -85,B 0,C 180,E1 -9912.904,E2 -9912.904} C_VEL
LIN {X 0,Y 425.359,Z 135.502,A -85,B 0,C 180,E1 -9916.605,E2 -9916.605} C_VEL
LIN {X 0,Y 425.326,Z 135.502,A -85,B 0,C 180,E1 -9919.636,E2 -9919.636} C_VEL
LIN {X 0,Y 425.304,Z 135.51,A -85,B 0,C 180,E1 -9923.365,E2 -9923.365} C_VEL
LIN {X 0,Y 425.346,Z 135.507,A -85,B 0,C 180,E1 -9926.844,E2 -9926.844} C_VEL
LIN {X 0,Y 425.289,Z 135.509,A -85,B 0,C 180,E1 -9929.72,E2 -9929.72} C_VEL
LIN {X 0,Y 425.323,Z 135.56,A -85,B 0,C 180,E1 -9932.14,E2 -9932.14} C_VEL
LIN {X 0,Y 427.102,Z 144.25,A -85,B 0,C 180,E1 -9934.187,E2 -9934.187} C_VEL
LIN {X 0,Y 430.452,Z 157.639,A -85,B 0,C 180,E1 -9934.602,E2 -9934.602} C_VEL
LIN {X 0,Y 431.167,Z 162.588,A -85,B 0,C 180,E1 -9934.729,E2 -9934.729} C_VEL
LIN {X 0,Y 429.969,Z 251.342,A -85,B 0,C 180,E1 -9936.306,E2 -9936.306} C_VEL
LIN {X 0,Y 429.575,Z 265.096,A -85,B 0,C 180,E1 -9936.75,E2 -9936.75} C_VEL
LIN {X 0,Y 429.171,Z 277.738,A -85,B 0,C 180,E1 -9937.362,E2 -9937.362} C_VEL
LIN {X 0,Y 428.558,Z 290.037,A -85,B 0,C 180,E1 -9938.174,E2 -9938.174} C_VEL
LIN {X 0,Y 427.995,Z 300.501,A -85,B 0,C 180,E1 -9939.057,E2 -9939.057} C_VEL
LIN {X 0,Y 427.289,Z 310.129,A -85,B 0,C 180,E1 -9940.055,E2 -9940.055} C_VEL
LIN {X 0,Y 426.66,Z 319.25,A -85,B 0,C 180,E1 -9941.215,E2 -9941.215} C_VEL
LIN {X 0,Y 425.966,Z 327.851,A -85,B 0,C 180,E1 -9942.567,E2 -9942.567} C_VEL
LIN {X 0,Y 425.446,Z 334.878,A -85,B 0,C 180,E1 -9943.932,E2 -9943.932} C_VEL
LIN {X 0,Y 425.06,Z 340.618,A -85,B 0,C 180,E1 -9945.314,E2 -9945.314} C_VEL
LIN {X 0,Y 424.771,Z 345.253,A -85,B 0,C 180,E1 -9946.718,E2 -9946.718} C_VEL
LIN {X 0,Y 424.492,Z 348.908,A -85,B 0,C 180,E1 -9948.162,E2 -9948.162} C_VEL
LIN {X 0,Y 424.275,Z 351.756,A -85,B 0,C 180,E1 -9949.758,E2 -9949.758} C_VEL
LIN {X 0,Y 424.163,Z 353.26,A -85,B 0,C 180,E1 -9951.146,E2 -9951.146} C_VEL
LIN {X 0,Y 424.1,Z 353.938,A -85,B 0,C 180,E1 -9952.696,E2 -9952.696} C_VEL
LIN {X 0,Y 424.115,Z 353.378,A -85,B 0,C 180,E1 -9954.551,E2 -9954.551} C_VEL
LIN {X 0,Y 424.193,Z 351.949,A -85,B 0,C 180,E1 -9955.934,E2 -9955.934} C_VEL
LIN {X 0,Y 424.402,Z 349.006,A -85,B 0,C 180,E1 -9957.623,E2 -9957.623} C_VEL
LIN {X 0,Y 424.679,Z 344.454,A -85,B 0,C 180,E1 -9959.378,E2 -9959.378} C_VEL
LIN {X 0,Y 424.987,Z 339.675,A -85,B 0,C 180,E1 -9960.762,E2 -9960.762} C_VEL
LIN {X 0,Y 425.392,Z 333.543,A -85,B 0,C 180,E1 -9962.178,E2 -9962.178} C_VEL
LIN {X 0,Y 425.848,Z 326.258,A -85,B 0,C 180,E1 -9963.539,E2 -9963.539} C_VEL
LIN {X 0,Y 426.427,Z 317.524,A -85,B 0,C 180,E1 -9964.853,E2 -9964.853} C_VEL
LIN {X 0,Y 427.119,Z 307.286,A -85,B 0,C 180,E1 -9966.097,E2 -9966.097} C_VEL
LIN {X 0,Y 427.7,Z 297.394,A -85,B 0,C 180,E1 -9967.071,E2 -9967.071} C_VEL
LIN {X 0,Y 428.3,Z 286.157,A -85,B 0,C 180,E1 -9967.954,E2 -9967.954} C_VEL
LIN {X 0,Y 428.818,Z 273.098,A -85,B 0,C 180,E1 -9968.74,E2 -9968.74} C_VEL
LIN {X 0,Y 429.243,Z 260.659,A -85,B 0,C 180,E1 -9969.28,E2 -9969.28} C_VEL
LIN {X 0,Y 429.54,Z 246.825,A -85,B 0,C 180,E1 -9969.661,E2 -9969.661} C_VEL
LIN {X 0,Y 429.816,Z 220.738,A -85,B 0,C 180,E1 -9970.117,E2 -9970.117} C_VEL
LIN {X 0,Y 429.287,Z 214.932,A -85,B 0,C 180,E1 -9970.24,E2 -9970.24} C_VEL
LIN {X 0,Y 424.08,Z 196.224,A -85,B 0,C 180,E1 -9970.783,E2 -9970.783} C_VEL
LIN {X 0,Y 423.437,Z 190.42,A -85,B 0,C 180,E1 -9970.915,E2 -9970.915} C_VEL
LIN {X 0,Y 423.662,Z 161.314,A -85,B 0,C 180,E1 -9971.439,E2 -9971.439} C_VEL
LIN {X 0,Y 420.13,Z 145.356,A -85,B 0,C 180,E1 -9971.887,E2 -9971.887} C_VEL
LIN {X 0,Y 419.625,Z 143.562,A -85,B 0,C 180,E1 -9971.951,E2 -9971.951} C_VEL
LIN {X 0,Y 418.373,Z 136.373,A -85,B 0,C 180,E1 -9973.721,E2 -9973.721} C_VEL
LIN {X 0,Y 418.355,Z 136.376,A -85,B 0,C 180,E1 -9977.386,E2 -9977.386} C_VEL
LIN {X 0,Y 418.4,Z 136.367,A -85,B 0,C 180,E1 -9981.305,E2 -9981.305} C_VEL
LIN {X 0,Y 418.509,Z 136.35,A -85,B 0,C 180,E1 -9984.217,E2 -9984.217} C_VEL
LIN {X 0,Y 418.541,Z 136.346,A -85,B 0,C 180,E1 -9988.076,E2 -9988.076} C_VEL
LIN {X 0,Y 418.671,Z 136.33,A -85,B 0,C 180,E1 -9990,E2 -9990} C_VEL
LIN {X 0,Y 418.501,Z 136.354,A -85,B 0,C 180,E1 -9992.888,E2 -9992.888} C_VEL
LIN {X 0,Y 418.5,Z 136.352,A -85,B 0,C 180,E1 -9995.783,E2 -9995.783} C_VEL
LIN {X 0,Y 418.377,Z 136.368,A -85,B 0,C 180,E1 -9998.696,E2 -9998.696} C_VEL
LIN {X 0,Y 418.315,Z 136.375,A -85,B 0,C 180,E1 -10001.631,E2 -10001.631} C_VEL
LIN {X 0,Y 418.303,Z 136.378,A -85,B 0,C 180,E1 -10004.597,E2 -10004.597} C_VEL
LIN {X 0,Y 418.28,Z 136.379,A -85,B 0,C 180,E1 -10007.604,E2 -10007.604} C_VEL
LIN {X 0,Y 418.249,Z 136.387,A -85,B 0,C 180,E1 -10010.663,E2 -10010.663} C_VEL
LIN {X 0,Y 418.276,Z 136.379,A -85,B 0,C 180,E1 -10013.782,E2 -10013.782} C_VEL
LIN {X 0,Y 418.309,Z 136.377,A -85,B 0,C 180,E1 -10017.07,E2 -10017.07} C_VEL
LIN {X 0,Y 418.243,Z 136.386,A -85,B 0,C 180,E1 -10020.272,E2 -10020.272} C_VEL
LIN {X 0,Y 418.246,Z 136.383,A -85,B 0,C 180,E1 -10023.677,E2 -10023.677} C_VEL
LIN {X 0,Y 418.238,Z 136.384,A -85,B 0,C 180,E1 -10027.224,E2 -10027.224} C_VEL
LIN {X 0,Y 418.243,Z 136.384,A -85,B 0,C 180,E1 -10029.683,E2 -10029.683} C_VEL
LIN {X 0,Y 418.228,Z 136.392,A -85,B 0,C 180,E1 -10032.321,E2 -10032.321} C_VEL
LIN {X 0,Y 418.236,Z 136.384,A -85,B 0,C 180,E1 -10035.109,E2 -10035.109} C_VEL
LIN {X 0,Y 418.239,Z 136.386,A -85,B 0,C 180,E1 -10037.767,E2 -10037.767} C_VEL
LIN {X 0,Y 418.258,Z 136.383,A -85,B 0,C 180,E1 -10040.618,E2 -10040.618} C_VEL
LIN {X 0,Y 418.244,Z 136.39,A -85,B 0,C 180,E1 -10043.976,E2 -10043.976} C_VEL
LIN {X 0,Y 418.256,Z 136.382,A -85,B 0,C 180,E1 -10047.156,E2 -10047.156} C_VEL
LIN {X 0,Y 418.267,Z 136.38,A -85,B 0,C 180,E1 -10050.895,E2 -10050.895} C_VEL
LIN {X 0,Y 418.266,Z 136.383,A -85,B 0,C 180,E1 -10054.096,E2 -10054.096} C_VEL
LIN {X 0,Y 418.23,Z 136.387,A -85,B 0,C 180,E1 -10057.264,E2 -10057.264} C_VEL
LIN {X 0,Y 418.281,Z 136.378,A -85,B 0,C 180,E1 -10060.364,E2 -10060.364} C_VEL
LIN {X 0,Y 418.315,Z 136.38,A -85,B 0,C 180,E1 -10063.405,E2 -10063.405} C_VEL
LIN {X 0,Y 418.345,Z 136.373,A -85,B 0,C 180,E1 -10066.999,E2 -10066.999} C_VEL
LIN {X 0,Y 418.34,Z 136.371,A -85,B 0,C 180,E1 -10070.329,E2 -10070.329} C_VEL
LIN {X 0,Y 418.512,Z 136.349,A -85,B 0,C 180,E1 -10072.28,E2 -10072.28} C_VEL
LIN {X 0,Y 418.513,Z 136.349,A -85,B 0,C 180,E1 -10074.217,E2 -10074.217} C_VEL
LIN {X 0,Y 418.543,Z 136.345,A -85,B 0,C 180,E1 -10078.076,E2 -10078.076} C_VEL
LIN {X 0,Y 418.671,Z 136.329,A -85,B 0,C 180,E1 -10080,E2 -10080} C_VEL
LIN {X 0,Y 418.509,Z 136.355,A -85,B 0,C 180,E1 -10082.888,E2 -10082.888} C_VEL
LIN {X 0,Y 418.486,Z 136.358,A -85,B 0,C 180,E1 -10086.751,E2 -10086.751} C_VEL
LIN {X 0,Y 418.34,Z 136.371,A -85,B 0,C 180,E1 -10089.672,E2 -10089.672} C_VEL
LIN {X 0,Y 418.345,Z 136.375,A -85,B 0,C 180,E1 -10093.001,E2 -10093.001} C_VEL
LIN {X 0,Y 418.312,Z 136.381,A -85,B 0,C 180,E1 -10096.736,E2 -10096.736} C_VEL
LIN {X 0,Y 418.27,Z 136.38,A -85,B 0,C 180,E1 -10099.791,E2 -10099.791} C_VEL
LIN {X 0,Y 418.231,Z 136.389,A -85,B 0,C 180,E1 -10102.737,E2 -10102.737} C_VEL
LIN {X 0,Y 418.27,Z 136.381,A -85,B 0,C 180,E1 -10105.904,E2 -10105.904} C_VEL
LIN {X 0,Y 418.264,Z 136.38,A -85,B 0,C 180,E1 -10109.162,E2 -10109.162} C_VEL
LIN {X 0,Y 418.257,Z 136.382,A -85,B 0,C 180,E1 -10112.844,E2 -10112.844} C_VEL
LIN {X 0,Y 418.248,Z 136.389,A -85,B 0,C 180,E1 -10116.239,E2 -10116.239} C_VEL
LIN {X 0,Y 418.265,Z 136.383,A -85,B 0,C 180,E1 -10119.681,E2 -10119.681} C_VEL
LIN {X 0,Y 418.246,Z 136.386,A -85,B 0,C 180,E1 -10122.324,E2 -10122.324} C_VEL
LIN {X 0,Y 418.236,Z 136.384,A -85,B 0,C 180,E1 -10125.109,E2 -10125.109} C_VEL
LIN {X 0,Y 418.257,Z 136.387,A -85,B 0,C 180,E1 -10127.769,E2 -10127.769} C_VEL
LIN {X 0,Y 418.268,Z 136.38,A -85,B 0,C 180,E1 -10130.617,E2 -10130.617} C_VEL
LIN {X 0,Y 418.247,Z 136.387,A -85,B 0,C 180,E1 -10133.976,E2 -10133.976} C_VEL
LIN {X 0,Y 418.259,Z 136.383,A -85,B 0,C 180,E1 -10137.156,E2 -10137.156} C_VEL
LIN {X 0,Y 418.27,Z 136.385,A -85,B 0,C 180,E1 -10140.896,E2 -10140.896} C_VEL
LIN {X 0,Y 418.326,Z 136.516,A -85,B 0,C 180,E1 -10141.495,E2 -10141.495} C_VEL
LIN {X 0,Y 420.848,Z 148.763,A -85,B 0,C 180,E1 -10144.001,E2 -10144.001} C_VEL
LIN {X 0,Y 421.493,Z 152.994,A -85,B 0,C 180,E1 -10144.838,E2 -10144.838} C_VEL
LIN {X 0,Y 420.309,Z 170.994,A -85,B 0,C 180,E1 -10148.158,E2 -10148.158} C_VEL
LIN {X 0,Y 419.585,Z 184.943,A -85,B 0,C 180,E1 -10150.708,E2 -10150.708} C_VEL
LIN {X 0,Y 419.438,Z 186.938,A -85,B 0,C 180,E1 -10151.066,E2 -10151.066} C_VEL
LIN {X 0,Y 423.292,Z 214.705,A -85,B 0,C 180,E1 -10151.736,E2 -10151.736} C_VEL
LIN {X 0,Y 422.34,Z 296.078,A -85,B 0,C 180,E1 -10153.194,E2 -10153.194} C_VEL
LIN {X 0,Y 421.844,Z 309.107,A -85,B 0,C 180,E1 -10153.61,E2 -10153.61} C_VEL
LIN {X 0,Y 421.223,Z 321.756,A -85,B 0,C 180,E1 -10154.207,E2 -10154.207} C_VEL
LIN {X 0,Y 420.472,Z 333.835,A -85,B 0,C 180,E1 -10154.985,E2 -10154.985} C_VEL
LIN {X 0,Y 419.757,Z 345.391,A -85,B 0,C 180,E1 -10155.95,E2 -10155.95} C_VEL
LIN {X 0,Y 419.137,Z 354.907,A -85,B 0,C 180,E1 -10156.937,E2 -10156.937} C_VEL
LIN {X 0,Y 418.541,Z 364.33,A -85,B 0,C 180,E1 -10158.13,E2 -10158.13} C_VEL
LIN {X 0,Y 417.845,Z 373.552,A -85,B 0,C 180,E1 -10159.583,E2 -10159.583} C_VEL
LIN {X 0,Y 417.47,Z 380.986,A -85,B 0,C 180,E1 -10161.041,E2 -10161.041} C_VEL
LIN {X 0,Y 417.301,Z 386.028,A -85,B 0,C 180,E1 -10162.257,E2 -10162.257} C_VEL
LIN {X 0,Y 417.131,Z 391.029,A -85,B 0,C 180,E1 -10163.753,E2 -10163.753} C_VEL
LIN {X 0,Y 417.138,Z 394.654,A -85,B 0,C 180,E1 -10165.168,E2 -10165.168} C_VEL
LIN {X 0,Y 417.058,Z 396.575,A -85,B 0,C 180,E1 -10166.135,E2 -10166.135} C_VEL
LIN {X 0,Y 417.163,Z 398.056,A -85,B 0,C 180,E1 -10167.103,E2 -10167.103} C_VEL
LIN {X 0,Y 417.126,Z 399.084,A -85,B 0,C 180,E1 -10168.069,E2 -10168.069} C_VEL
LIN {X 0,Y 417.114,Z 399.715,A -85,B 0,C 180,E1 -10169.035,E2 -10169.035} C_VEL
LIN {X 0,Y 417.118,Z 399.953,A -85,B 0,C 180,E1 -10170,E2 -10170} C_VEL
LIN {X 0,Y 417.1,Z 399.767,A -85,B 0,C 180,E1 -10170.965,E2 -10170.965} C_VEL
LIN {X 0,Y 417.117,Z 399.156,A -85,B 0,C 180,E1 -10171.931,E2 -10171.931} C_VEL
LIN {X 0,Y 417.131,Z 398.149,A -85,B 0,C 180,E1 -10172.897,E2 -10172.897} C_VEL
LIN {X 0,Y 417.056,Z 396.736,A -85,B 0,C 180,E1 -10173.865,E2 -10173.865} C_VEL
LIN {X 0,Y 417.127,Z 393.771,A -85,B 0,C 180,E1 -10175.317,E2 -10175.317} C_VEL
LIN {X 0,Y 417.159,Z 389.756,A -85,B 0,C 180,E1 -10176.773,E2 -10176.773} C_VEL
LIN {X 0,Y 417.434,Z 383.609,A -85,B 0,C 180,E1 -10178.471,E2 -10178.471} C_VEL
LIN {X 0,Y 417.763,Z 376.878,A -85,B 0,C 180,E1 -10179.929,E2 -10179.929} C_VEL
LIN {X 0,Y 418.329,Z 368.54,A -85,B 0,C 180,E1 -10181.385,E2 -10181.385} C_VEL
LIN {X 0,Y 418.891,Z 360.027,A -85,B 0,C 180,E1 -10182.598,E2 -10182.598} C_VEL
LIN {X 0,Y 419.621,Z 349.781,A -85,B 0,C 180,E1 -10183.783,E2 -10183.783} C_VEL
LIN {X 0,Y 420.453,Z 337.755,A -85,B 0,C 180,E1 -10184.892,E2 -10184.892} C_VEL
LIN {X 0,Y 421.268,Z 326.047,A -85,B 0,C 180,E1 -10185.729,E2 -10185.729} C_VEL
LIN {X 0,Y 422.047,Z 312.636,A -85,B 0,C 180,E1 -10186.444,E2 -10186.444} C_VEL
LIN {X 0,Y 422.673,Z 299.922,A -85,B 0,C 180,E1 -10186.917,E2 -10186.917} C_VEL
LIN {X 0,Y 423.009,Z 285.084,A -85,B 0,C 180,E1 -10187.245,E2 -10187.245} C_VEL
LIN {X 0,Y 423.76,Z 214.058,A -85,B 0,C 180,E1 -10188.517,E2 -10188.517} C_VEL
LIN {X 0,Y 420.686,Z 192.142,A -85,B 0,C 180,E1 -10189.078,E2 -10189.078} C_VEL
LIN {X 0,Y 419.591,Z 185.379,A -85,B 0,C 180,E1 -10189.292,E2 -10189.292} C_VEL
LIN {X 0,Y 420.76,Z 165.252,A -85,B 0,C 180,E1 -10192.948,E2 -10192.948} C_VEL
LIN {X 0,Y 421.551,Z 152.25,A -85,B 0,C 180,E1 -10195.348,E2 -10195.348} C_VEL
LIN {X 0,Y 419.391,Z 141.082,A -85,B 0,C 180,E1 -10197.618,E2 -10197.618} C_VEL
LIN {X 0,Y 418.313,Z 136.383,A -85,B 0,C 180,E1 -10198.608,E2 -10198.608} C_VEL
LIN {X 0,Y 418.213,Z 136.39,A -85,B 0,C 180,E1 -10201.396,E2 -10201.396} C_VEL
LIN {X 0,Y 418.266,Z 136.388,A -85,B 0,C 180,E1 -10204.58,E2 -10204.58} C_VEL
LIN {X 0,Y 418.238,Z 136.391,A -85,B 0,C 180,E1 -10207.835,E2 -10207.835} C_VEL
LIN {X 0,Y 418.266,Z 136.384,A -85,B 0,C 180,E1 -10210.942,E2 -10210.942} C_VEL
LIN {X 0,Y 418.21,Z 136.393,A -85,B 0,C 180,E1 -10213.729,E2 -10213.729} C_VEL
LIN {X 0,Y 418.209,Z 136.394,A -85,B 0,C 180,E1 -10216.448,E2 -10216.448} C_VEL
LIN {X 0,Y 418.265,Z 136.382,A -85,B 0,C 180,E1 -10219.123,E2 -10219.123} C_VEL
LIN {X 0,Y 418.237,Z 136.39,A -85,B 0,C 180,E1 -10222.165,E2 -10222.165} C_VEL
LIN {X 0,Y 418.265,Z 136.383,A -85,B 0,C 180,E1 -10225.419,E2 -10225.419} C_VEL
LIN {X 0,Y 418.21,Z 136.389,A -85,B 0,C 180,E1 -10228.604,E2 -10228.604} C_VEL
LIN {X 0,Y 418.29,Z 136.381,A -85,B 0,C 180,E1 -10231.936,E2 -10231.936} C_VEL
LIN {X 0,Y 418.289,Z 136.377,A -85,B 0,C 180,E1 -10235.162,E2 -10235.162} C_VEL
LIN {X 0,Y 418.233,Z 136.383,A -85,B 0,C 180,E1 -10238.303,E2 -10238.303} C_VEL
LIN {X 0,Y 418.282,Z 136.377,A -85,B 0,C 180,E1 -10241.383,E2 -10241.383} C_VEL
LIN {X 0,Y 418.301,Z 136.373,A -85,B 0,C 180,E1 -10244.406,E2 -10244.406} C_VEL
